// Mitsubishi GX Works2 project: UNLD LINE 4   PLC: Q06UDV

PROGRAM DATALINK
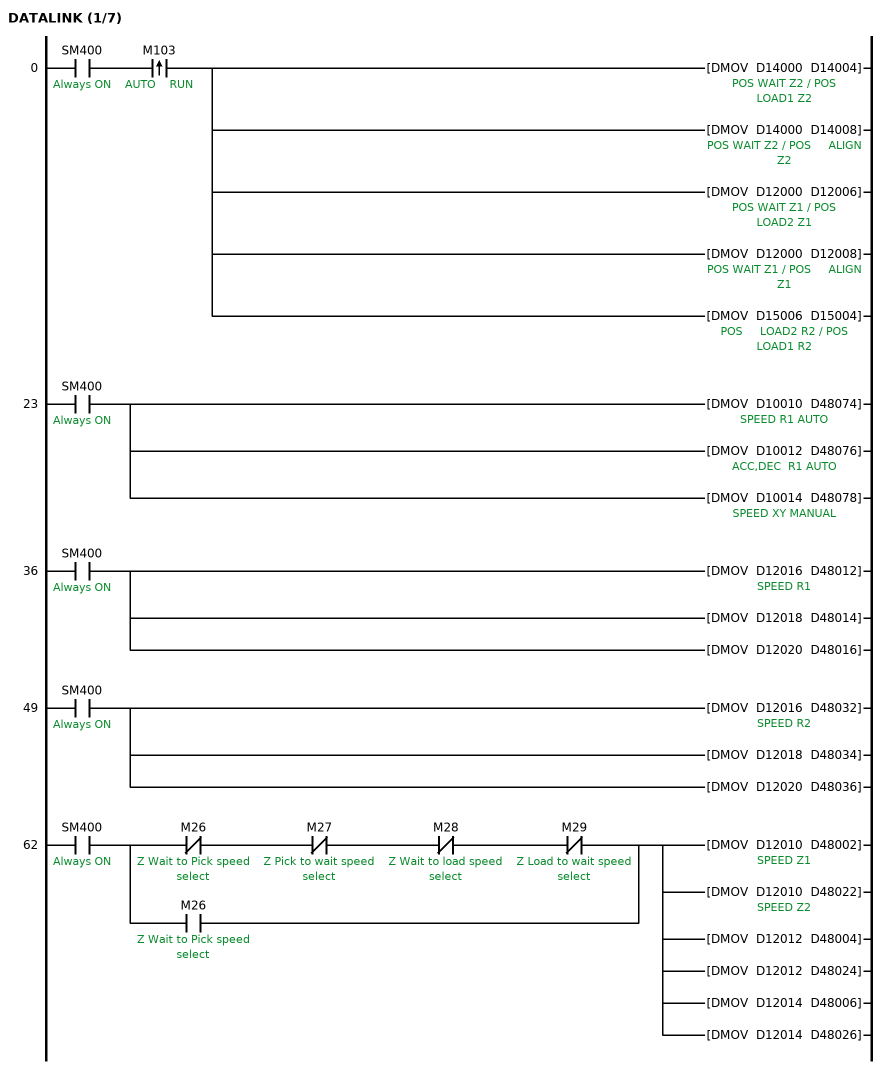
0     LD      SM400  ; Always ON
      ANDP    M103  ; AUTO    RUN
      DMOV    D14000 D14004  ; POS WAIT Z2 / POS     LOAD1 Z2
      DMOV    D14000 D14008  ; POS     ALIGN Z2
      DMOV    D12000 D12006  ; POS WAIT Z1 / POS     LOAD2 Z1
      DMOV    D12000 D12008  ; POS     ALIGN Z1
      DMOV    D15006 D15004  ; POS     LOAD2 R2 / POS     LOAD1 R2
23    LD      SM400  ; Always ON
      DMOV    D10010 D48074  ; SPEED R1 AUTO
      DMOV    D10012 D48076  ; ACC,DEC  R1 AUTO
      DMOV    D10014 D48078  ; SPEED XY MANUAL
36    LD      SM400  ; Always ON
      DMOV    D12016 D48012  ; SPEED R1
      DMOV    D12018 D48014
      DMOV    D12020 D48016
49    LD      SM400  ; Always ON
      DMOV    D12016 D48032  ; SPEED R2
      DMOV    D12018 D48034
      DMOV    D12020 D48036
62    LD      SM400  ; Always ON
      LDI     M26  ; Z Wait to Pick speed select
      ANI     M27  ; Z Pick to wait speed select
      ANI     M28  ; Z Wait to load speed select
      ANI     M29  ; Z Load to wait speed select
      OR      M26  ; Z Wait to Pick speed select
      ANB
      DMOV    D12010 D48002  ; SPEED Z1
      DMOV    D12010 D48022  ; SPEED Z2
      DMOV    D12012 D48004
      DMOV    D12012 D48024
      DMOV    D12014 D48006
      DMOV    D12014 D48026
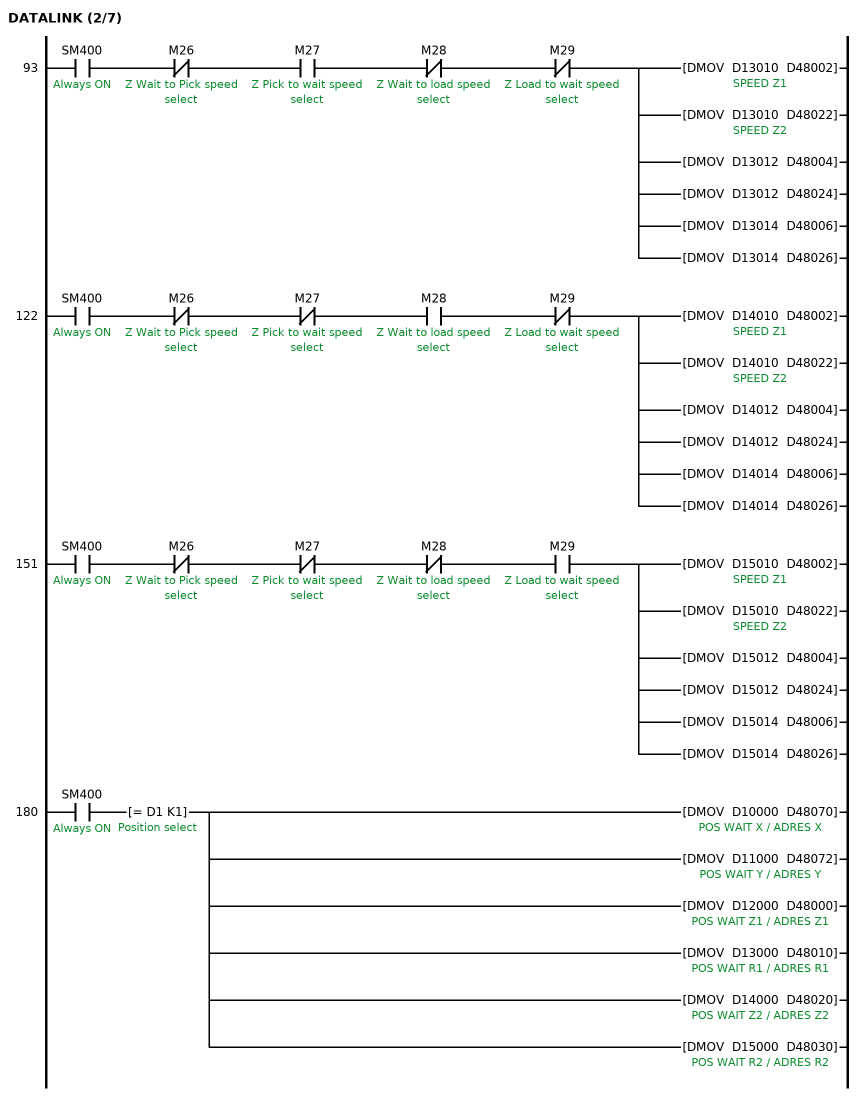
93    LD      SM400  ; Always ON
      ANI     M26  ; Z Wait to Pick speed select
      AND     M27  ; Z Pick to wait speed select
      ANI     M28  ; Z Wait to load speed select
      ANI     M29  ; Z Load to wait speed select
      DMOV    D13010 D48002
      DMOV    D13010 D48022
      DMOV    D13012 D48004
      DMOV    D13012 D48024
      DMOV    D13014 D48006
      DMOV    D13014 D48026
122   LD      SM400  ; Always ON
      ANI     M26  ; Z Wait to Pick speed select
      ANI     M27  ; Z Pick to wait speed select
      AND     M28  ; Z Wait to load speed select
      ANI     M29  ; Z Load to wait speed select
      DMOV    D14010 D48002
      DMOV    D14010 D48022
      DMOV    D14012 D48004
      DMOV    D14012 D48024
      DMOV    D14014 D48006
      DMOV    D14014 D48026
151   LD      SM400  ; Always ON
      ANI     M26  ; Z Wait to Pick speed select
      ANI     M27  ; Z Pick to wait speed select
      ANI     M28  ; Z Wait to load speed select
      AND     M29  ; Z Load to wait speed select
      DMOV    D15010 D48002
      DMOV    D15010 D48022
      DMOV    D15012 D48004
      DMOV    D15012 D48024
      DMOV    D15014 D48006
      DMOV    D15014 D48026
180   LD      SM400  ; Always ON
      AND=    D1 K1  ; Position select
      DMOV    D10000 D48070  ; POS WAIT X / ADRES X
      DMOV    D11000 D48072  ; POS WAIT Y / ADRES Y
      DMOV    D12000 D48000  ; ADRES Z1
      DMOV    D13000 D48010  ; POS WAIT R1 / ADRES R1
      DMOV    D14000 D48020  ; ADRES Z2
      DMOV    D15000 D48030  ; POS WAIT R2 / ADRES R2
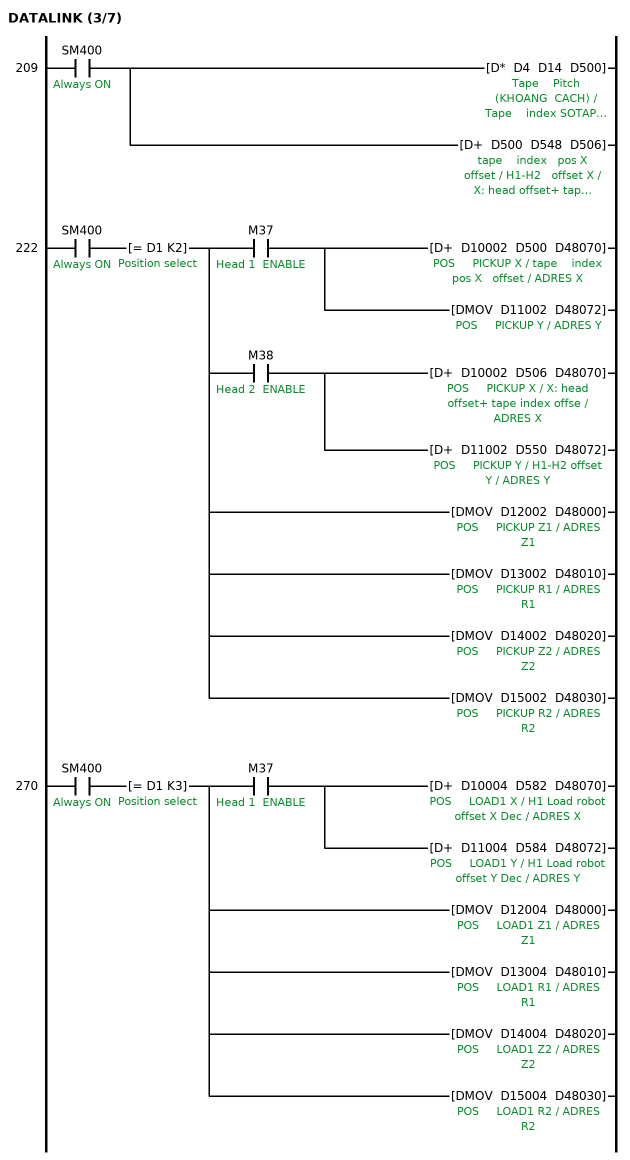
209   LD      SM400  ; Always ON
      D*      D4 D14 D500  ; Tape    Pitch   (KHOANG  CACH) / Tape    index SOTAPE HUT DUOC / tape    index   pos X   offset
      D+      D500 D548 D506  ; H1-H2   offset X / X: head offset+ tape index offse
222   LD      SM400  ; Always ON
      AND=    D1 K2  ; Position select
      MPS
      AND     M37  ; Head 1  ENABLE
      D+      D10002 D500 D48070  ; POS     PICKUP X
      DMOV    D11002 D48072  ; POS     PICKUP Y
      MRD
      AND     M38  ; Head 2  ENABLE
      D+      D10002 D506 D48070
      D+      D11002 D550 D48072  ; H1-H2 offset Y
      MPP
      DMOV    D12002 D48000  ; POS     PICKUP Z1
      DMOV    D13002 D48010  ; POS     PICKUP R1
      DMOV    D14002 D48020  ; POS     PICKUP Z2
      DMOV    D15002 D48030  ; POS     PICKUP R2
270   LD      SM400  ; Always ON
      AND=    D1 K3  ; Position select
      MPS
      AND     M37  ; Head 1  ENABLE
      D+      D10004 D582 D48070  ; POS     LOAD1 X / H1 Load robot offset X Dec
      D+      D11004 D584 D48072  ; POS     LOAD1 Y / H1 Load robot offset Y Dec
      MPP
      DMOV    D12004 D48000  ; POS     LOAD1 Z1
      DMOV    D13004 D48010  ; POS     LOAD1 R1
      DMOV    D14004 D48020
      DMOV    D15004 D48030
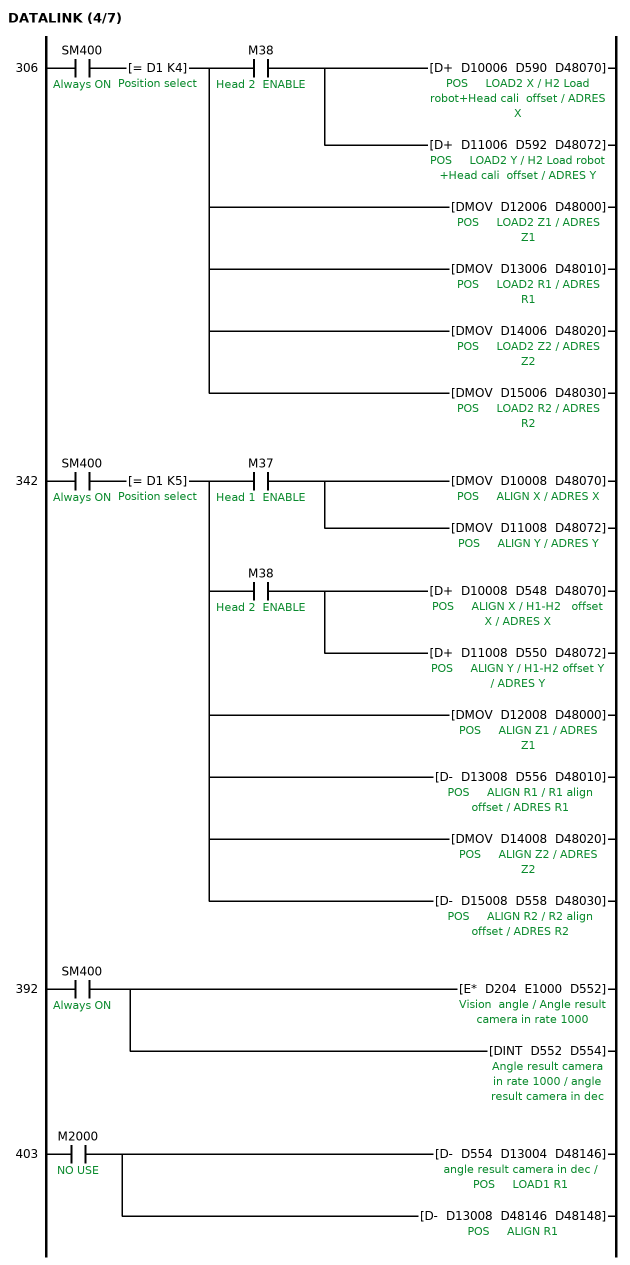
306   LD      SM400  ; Always ON
      AND=    D1 K4  ; Position select
      MPS
      AND     M38  ; Head 2  ENABLE
      D+      D10006 D590 D48070  ; POS     LOAD2 X / H2 Load robot+Head cali  offset
      D+      D11006 D592 D48072  ; POS     LOAD2 Y / H2 Load robot +Head cali  offset
      MPP
      DMOV    D12006 D48000
      DMOV    D13006 D48010  ; POS     LOAD2 R1
      DMOV    D14006 D48020  ; POS     LOAD2 Z2
      DMOV    D15006 D48030
342   LD      SM400  ; Always ON
      AND=    D1 K5  ; Position select
      MPS
      AND     M37  ; Head 1  ENABLE
      DMOV    D10008 D48070  ; POS     ALIGN X
      DMOV    D11008 D48072  ; POS     ALIGN Y
      MRD
      AND     M38  ; Head 2  ENABLE
      D+      D10008 D548 D48070
      D+      D11008 D550 D48072
      MPP
      DMOV    D12008 D48000
      D-      D13008 D556 D48010  ; POS     ALIGN R1 / R1 align offset
      DMOV    D14008 D48020
      D-      D15008 D558 D48030  ; POS     ALIGN R2 / R2 align offset
392   LD      SM400  ; Always ON
      E*      D204 E1000 D552  ; Vision  angle / Angle result camera in rate 1000
      DINT    D552 D554  ; angle result camera in dec
403   LD      M2000  ; NO USE
      D-      D554 D13004 D48146
      D-      D13008 D48146 D48148
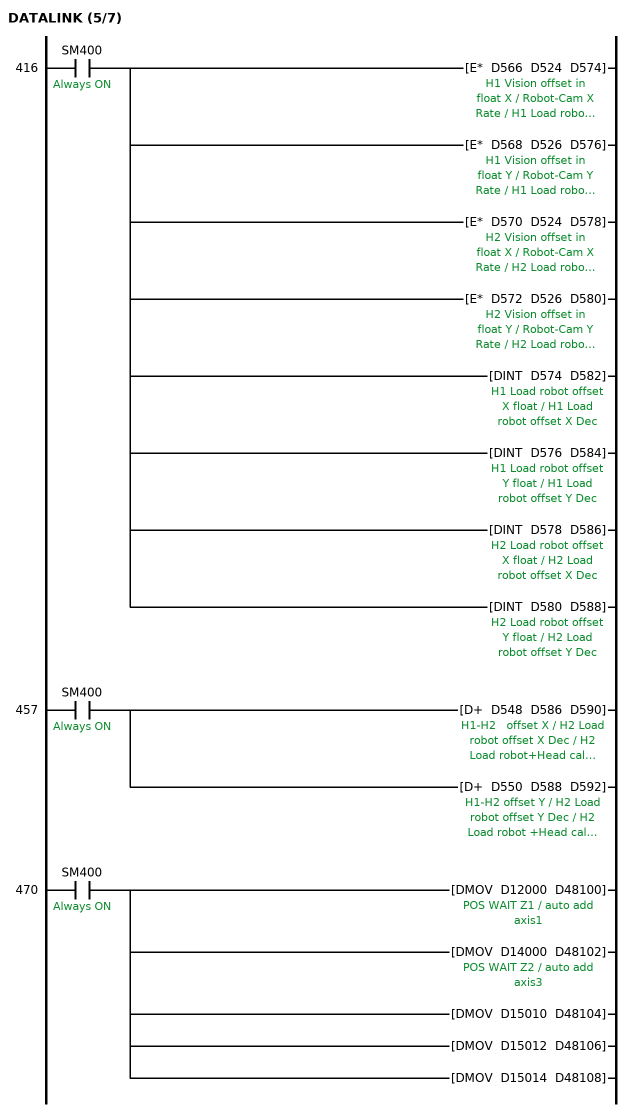
416   LD      SM400  ; Always ON
      E*      D566 D524 D574  ; H1 Vision offset in     float X / Robot-Cam X Rate / H1 Load robot offset X float
      E*      D568 D526 D576  ; H1 Vision offset in     float Y / Robot-Cam Y Rate / H1 Load robot offset Y float
      E*      D570 D524 D578  ; H2 Vision offset in     float X / H2 Load robot offset X float
      E*      D572 D526 D580  ; H2 Vision offset in     float Y / H2 Load robot offset Y float
      DINT    D574 D582
      DINT    D576 D584
      DINT    D578 D586  ; H2 Load robot offset X Dec
      DINT    D580 D588  ; H2 Load robot offset Y Dec
457   LD      SM400  ; Always ON
      D+      D548 D586 D590
      D+      D550 D588 D592
470   LD      SM400  ; Always ON
      DMOV    D12000 D48100  ; auto add axis1
      DMOV    D14000 D48102  ; auto add axis3
      DMOV    D15010 D48104
      DMOV    D15012 D48106
      DMOV    D15014 D48108
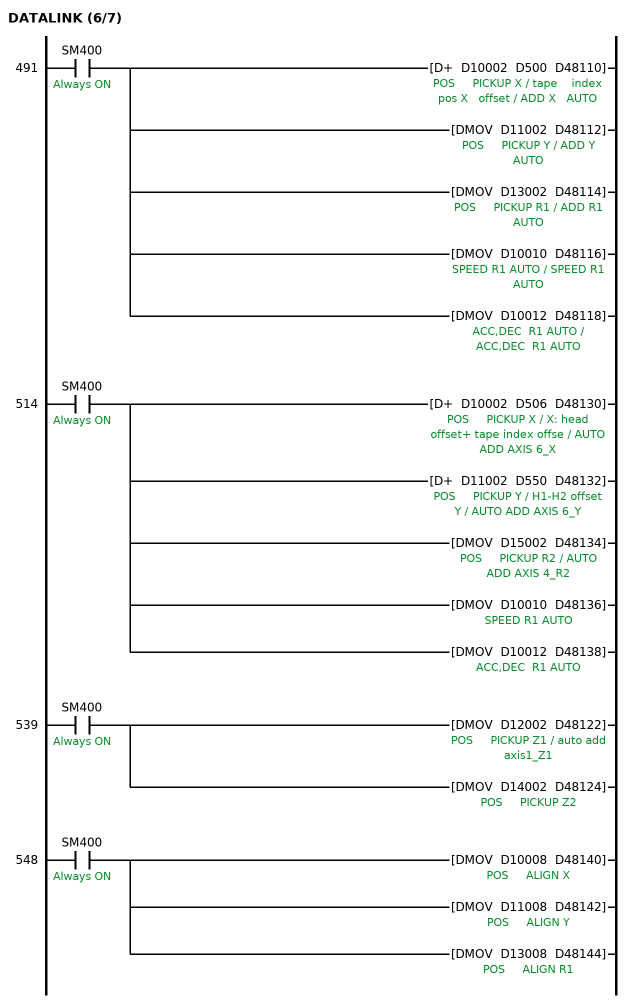
491   LD      SM400  ; Always ON
      D+      D10002 D500 D48110  ; ADD X   AUTO
      DMOV    D11002 D48112  ; ADD Y   AUTO
      DMOV    D13002 D48114  ; ADD R1  AUTO
      DMOV    D10010 D48116  ; SPEED R1 AUTO
      DMOV    D10012 D48118  ; ACC,DEC  R1 AUTO
514   LD      SM400  ; Always ON
      D+      D10002 D506 D48130  ; AUTO ADD AXIS 6_X
      D+      D11002 D550 D48132  ; AUTO ADD AXIS 6_Y
      DMOV    D15002 D48134  ; AUTO ADD AXIS 4_R2
      DMOV    D10010 D48136
      DMOV    D10012 D48138
539   LD      SM400  ; Always ON
      DMOV    D12002 D48122  ; auto add axis1_Z1
      DMOV    D14002 D48124
548   LD      SM400  ; Always ON
      DMOV    D10008 D48140
      DMOV    D11008 D48142
      DMOV    D13008 D48144
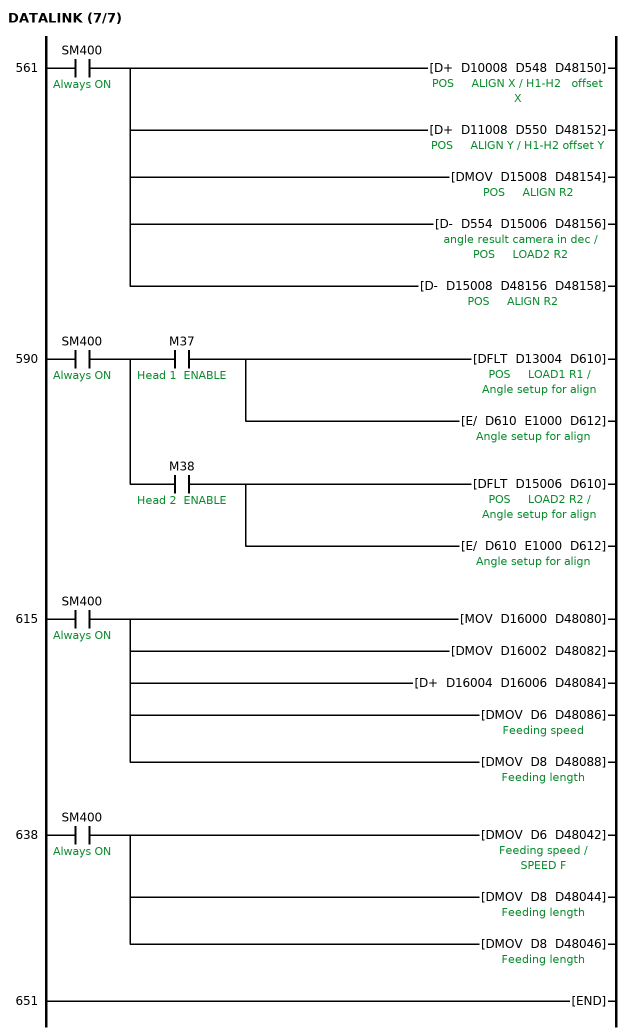
561   LD      SM400  ; Always ON
      D+      D10008 D548 D48150
      D+      D11008 D550 D48152
      DMOV    D15008 D48154
      D-      D554 D15006 D48156
      D-      D15008 D48156 D48158
590   LD      SM400  ; Always ON
      MPS
      AND     M37  ; Head 1  ENABLE
      DFLT    D13004 D610  ; Angle setup for align
      E/      D610 E1000 D612
      MPP
      AND     M38  ; Head 2  ENABLE
      DFLT    D15006 D610
      E/      D610 E1000 D612
615   LD      SM400  ; Always ON
      MOV     D16000 D48080
      DMOV    D16002 D48082
      D+      D16004 D16006 D48084
      DMOV    D6 D48086  ; Feeding speed
      DMOV    D8 D48088  ; Feeding length
638   LD      SM400  ; Always ON
      DMOV    D6 D48042  ; SPEED F
      DMOV    D8 D48044
      DMOV    D8 D48046
651   END
END_PROGRAM

PROGRAM MAIN
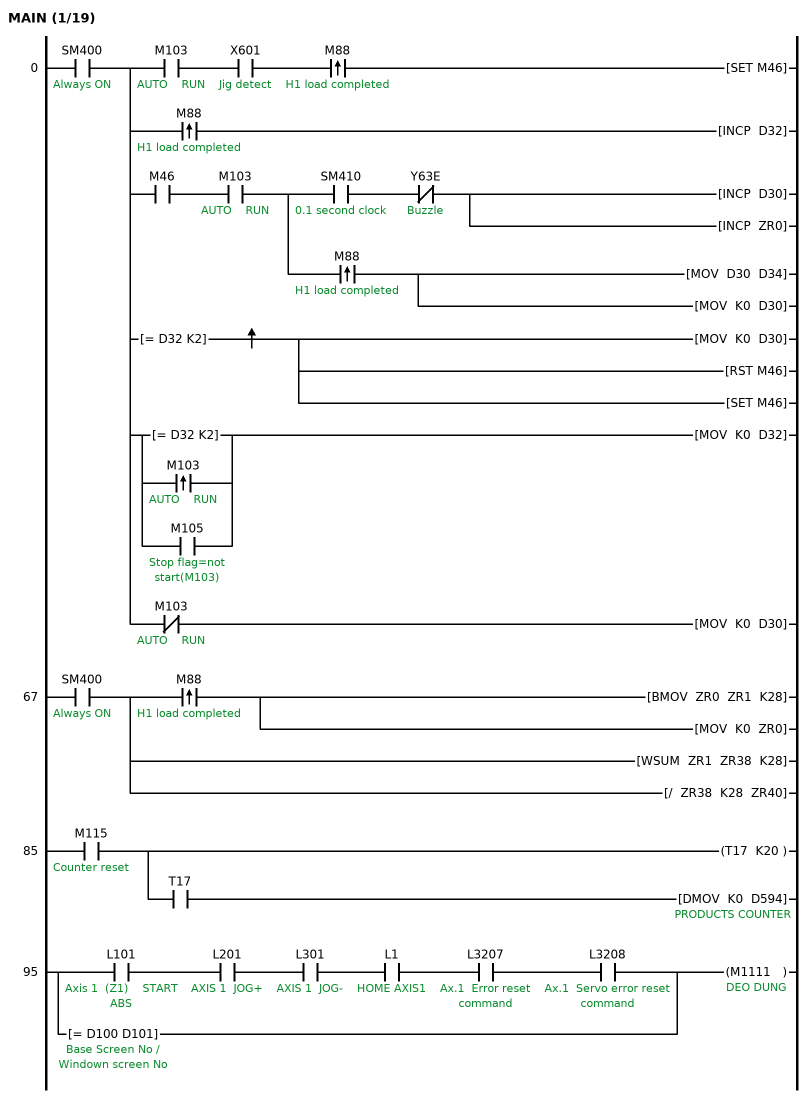
0     LD      SM400  ; Always ON
      MPS
      AND     M103  ; AUTO    RUN
      AND     X601  ; Jig detect
      ANDP    M88  ; H1 load completed
      SET     M46
      MRD
      ANDP    M88  ; H1 load completed
      INCP    D32
      MRD
      AND     M46
      AND     M103  ; AUTO    RUN
      MPS
      AND     SM410  ; 0.1 second clock
      ANI     Y63E  ; Buzzle
      INCP    D30
      INCP    ZR0
      MPP
      ANDP    M88  ; H1 load completed
      MOV     D30 D34
      MOV     K0 D30
      MRD
      AND=    D32 K2
      MEP
      MOV     K0 D30
      RST     M46
      SET     M46
      MRD
      LD=     D32 K2
      ORP     M103  ; AUTO    RUN
      OR      M105  ; Stop flag=not start(M103)
      ANB
      MOV     K0 D32
      MPP
      ANI     M103  ; AUTO    RUN
      MOV     K0 D30
67    LD      SM400  ; Always ON
      MPS
      ANDP    M88  ; H1 load completed
      BMOV    ZR0 ZR1 K28
      MOV     K0 ZR0
      MPP
      WSUM    ZR1 ZR38 K28
      /       ZR38 K28 ZR40
85    LD      M115  ; Counter reset
      OUT     T17 K20
      AND     T17
      DMOV    K0 D594  ; PRODUCTS COUNTER
95    LD      L101  ; Axis 1  (Z1)    START   ABS
      AND     L201  ; AXIS 1  JOG+
      AND     L301  ; AXIS 1  JOG-
      AND     L1  ; HOME AXIS1
      AND     L3207  ; Ax.1  Error reset command
      AND     L3208  ; Ax.1  Servo error reset command
      OR=     D100 D101  ; Base Screen No / Windown screen No
      OUT     M1111  ; DEO DUNG
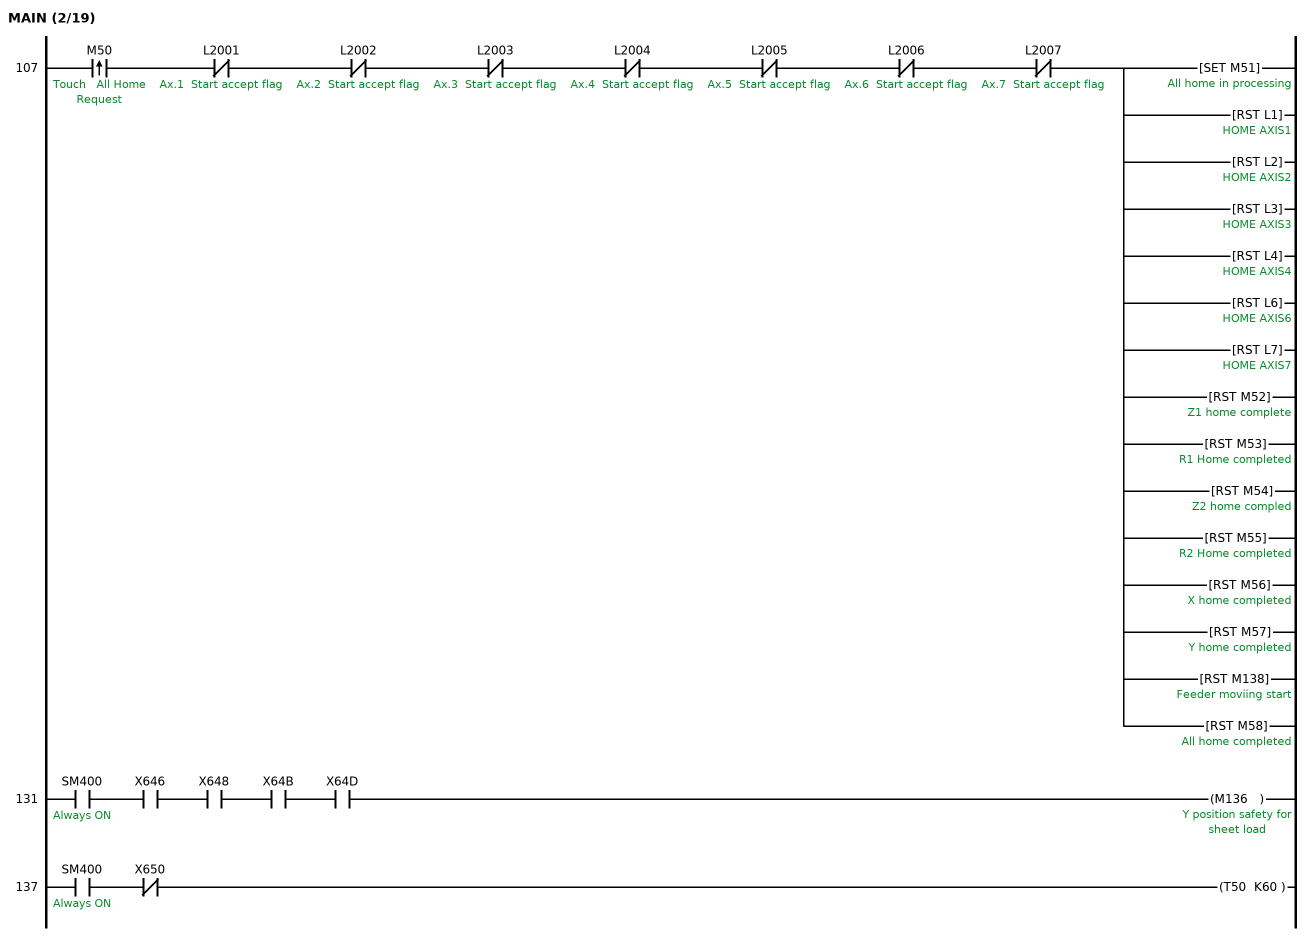
107   LDP     M50  ; Touch   All Home Request
      ANI     L2001  ; Ax.1  Start accept flag
      ANI     L2002  ; Ax.2  Start accept flag
      ANI     L2003  ; Ax.3  Start accept flag
      ANI     L2004  ; Ax.4  Start accept flag
      ANI     L2005  ; Ax.5  Start accept flag
      ANI     L2006  ; Ax.6  Start accept flag
      ANI     L2007  ; Ax.7  Start accept flag
      SET     M51  ; All home in processing
      RST     L1  ; HOME AXIS1
      RST     L2  ; HOME AXIS2
      RST     L3  ; HOME AXIS3
      RST     L4  ; HOME AXIS4
      RST     L6  ; HOME AXIS6
      RST     L7  ; HOME AXIS7
      RST     M52  ; Z1 home complete
      RST     M53  ; R1 Home completed
      RST     M54  ; Z2 home compled
      RST     M55  ; R2 Home completed
      RST     M56  ; X home completed
      RST     M57  ; Y home completed
      RST     M138  ; Feeder moviing start
      RST     M58  ; All home completed
131   LD      SM400  ; Always ON
      AND     X646
      AND     X648
      AND     X64B
      AND     X64D
      OUT     M136  ; Y position safety for sheet load
137   LD      SM400  ; Always ON
      ANI     X650
      OUT     T50 K60
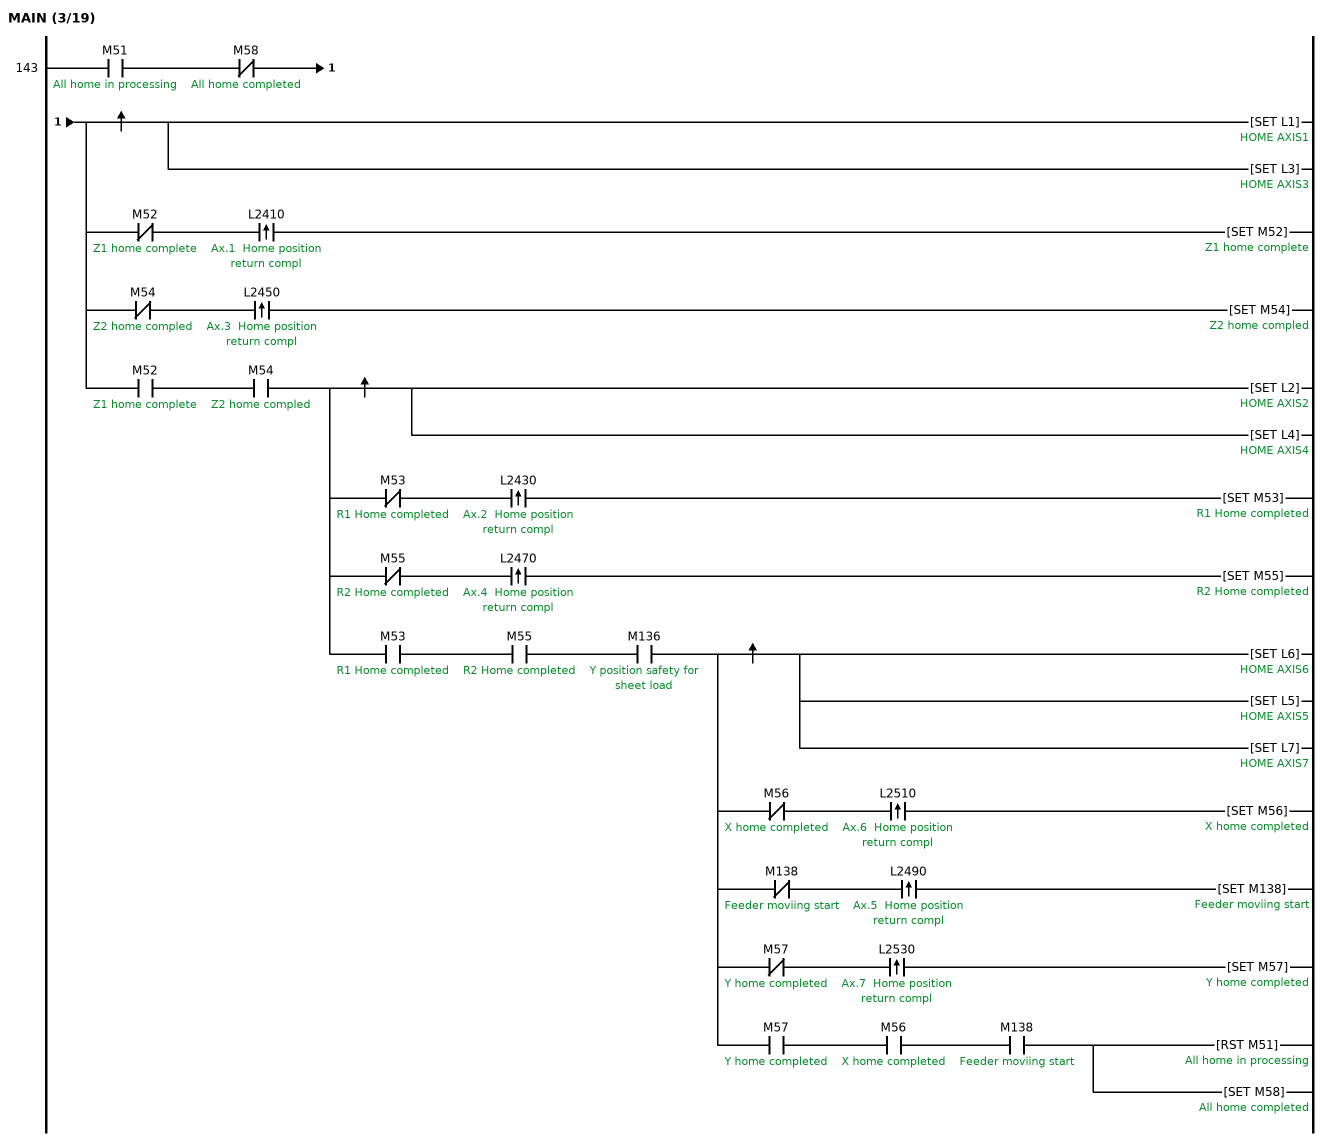
143   LD      M51  ; All home in processing
      ANI     M58  ; All home completed
      MPS
      MEP
      SET     L1  ; HOME AXIS1
      SET     L3  ; HOME AXIS3
      MRD
      ANI     M52  ; Z1 home complete
      ANDP    L2410  ; Ax.1  Home position return compl
      SET     M52  ; Z1 home complete
      MRD
      ANI     M54  ; Z2 home compled
      ANDP    L2450  ; Ax.3  Home position return compl
      SET     M54  ; Z2 home compled
      MPP
      AND     M52  ; Z1 home complete
      AND     M54  ; Z2 home compled
      MPS
      MEP
      SET     L2  ; HOME AXIS2
      SET     L4  ; HOME AXIS4
      MRD
      ANI     M53  ; R1 Home completed
      ANDP    L2430  ; Ax.2  Home position return compl
      SET     M53  ; R1 Home completed
      MRD
      ANI     M55  ; R2 Home completed
      ANDP    L2470  ; Ax.4  Home position return compl
      SET     M55  ; R2 Home completed
      MPP
      AND     M53  ; R1 Home completed
      AND     M55  ; R2 Home completed
      AND     M136  ; Y position safety for sheet load
      MPS
      MEP
      SET     L6  ; HOME AXIS6
      SET     L5  ; HOME AXIS5
      SET     L7  ; HOME AXIS7
      MRD
      ANI     M56  ; X home completed
      ANDP    L2510  ; Ax.6  Home position return compl
      SET     M56  ; X home completed
      MRD
      ANI     M138  ; Feeder moviing start
      ANDP    L2490  ; Ax.5  Home position return compl
      SET     M138  ; Feeder moviing start
      MRD
      ANI     M57  ; Y home completed
      ANDP    L2530  ; Ax.7  Home position return compl
      SET     M57  ; Y home completed
      MPP
      AND     M57  ; Y home completed
      AND     M56  ; X home completed
      AND     M138  ; Feeder moviing start
      RST     M51  ; All home in processing
      SET     M58  ; All home completed
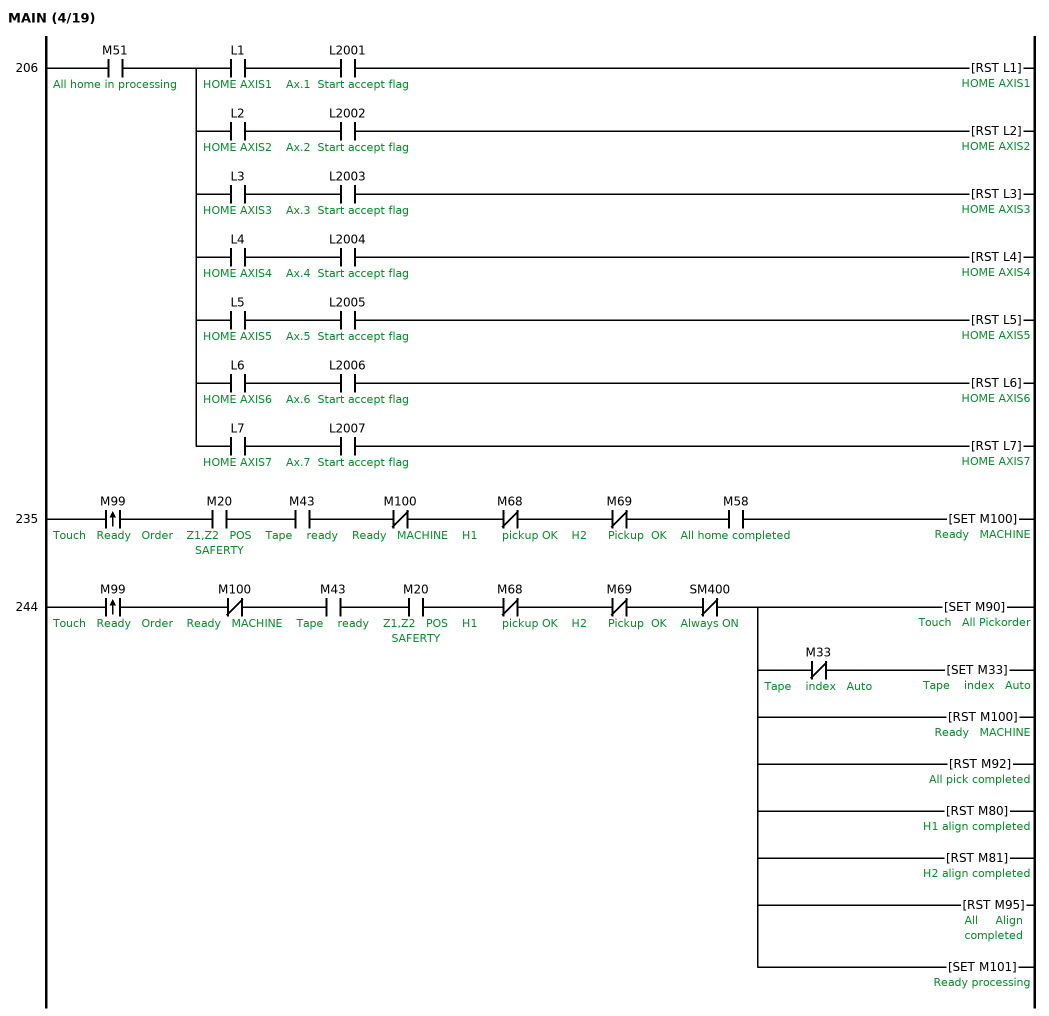
206   LD      M51  ; All home in processing
      MPS
      AND     L1  ; HOME AXIS1
      AND     L2001  ; Ax.1  Start accept flag
      RST     L1  ; HOME AXIS1
      MRD
      AND     L2  ; HOME AXIS2
      AND     L2002  ; Ax.2  Start accept flag
      RST     L2  ; HOME AXIS2
      MRD
      AND     L3  ; HOME AXIS3
      AND     L2003  ; Ax.3  Start accept flag
      RST     L3  ; HOME AXIS3
      MRD
      AND     L4  ; HOME AXIS4
      AND     L2004  ; Ax.4  Start accept flag
      RST     L4  ; HOME AXIS4
      MRD
      AND     L5  ; HOME AXIS5
      AND     L2005  ; Ax.5  Start accept flag
      RST     L5  ; HOME AXIS5
      MRD
      AND     L6  ; HOME AXIS6
      AND     L2006  ; Ax.6  Start accept flag
      RST     L6  ; HOME AXIS6
      MPP
      AND     L7  ; HOME AXIS7
      AND     L2007  ; Ax.7  Start accept flag
      RST     L7  ; HOME AXIS7
235   LDP     M99  ; Touch   Ready   Order
      AND     M20  ; Z1,Z2   POS     SAFERTY
      AND     M43  ; Tape    ready
      ANI     M100  ; Ready   MACHINE
      ANI     M68  ; H1       pickup OK
      ANI     M69  ; H2      Pickup  OK
      AND     M58  ; All home completed
      SET     M100  ; Ready   MACHINE
244   LDP     M99  ; Touch   Ready   Order
      ANI     M100  ; Ready   MACHINE
      AND     M43  ; Tape    ready
      AND     M20  ; Z1,Z2   POS     SAFERTY
      ANI     M68  ; H1       pickup OK
      ANI     M69  ; H2      Pickup  OK
      ANI     SM400  ; Always ON
      SET     M90  ; Touch   All Pickorder
      MPS
      ANI     M33  ; Tape    index   Auto
      SET     M33  ; Tape    index   Auto
      MPP
      RST     M100  ; Ready   MACHINE
      RST     M92  ; All pick completed
      RST     M80  ; H1 align completed
      RST     M81  ; H2 align completed
      RST     M95  ; All     Align   completed
      SET     M101  ; Ready processing
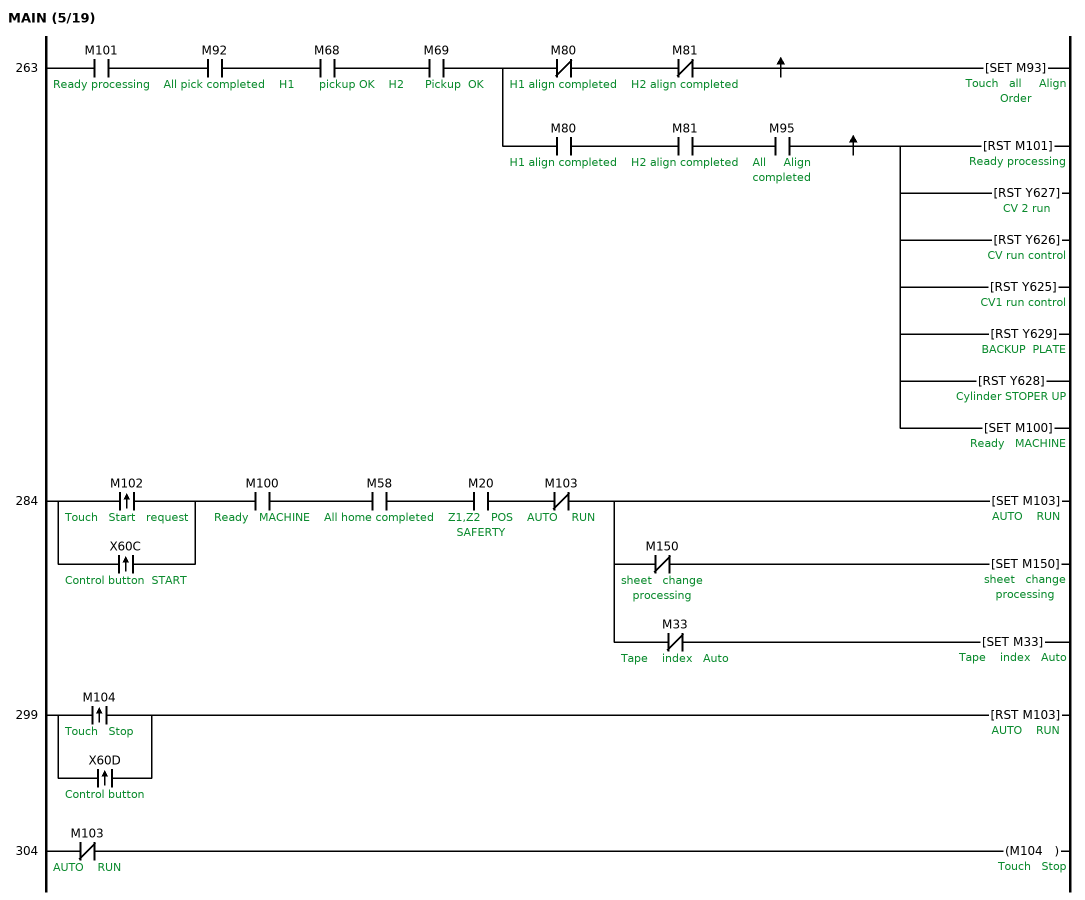
263   LD      M101  ; Ready processing
      AND     M92  ; All pick completed
      AND     M68  ; H1       pickup OK
      AND     M69  ; H2      Pickup  OK
      MPS
      ANI     M80  ; H1 align completed
      ANI     M81  ; H2 align completed
      MEP
      SET     M93  ; Touch   all     Align   Order
      MPP
      AND     M80  ; H1 align completed
      AND     M81  ; H2 align completed
      AND     M95  ; All     Align   completed
      MEP
      RST     M101  ; Ready processing
      RST     Y627  ; CV 2 run
      RST     Y626  ; CV run control
      RST     Y625  ; CV1 run control
      RST     Y629  ; BACKUP  PLATE
      RST     Y628  ; Cylinder STOPER UP
      SET     M100  ; Ready   MACHINE
284   LDP     M102  ; Touch   Start   request
      ORP     X60C  ; Control button  START
      AND     M100  ; Ready   MACHINE
      AND     M58  ; All home completed
      AND     M20  ; Z1,Z2   POS     SAFERTY
      ANI     M103  ; AUTO    RUN
      SET     M103  ; AUTO    RUN
      MPS
      ANI     M150  ; sheet   change  processing
      SET     M150  ; sheet   change  processing
      MPP
      ANI     M33  ; Tape    index   Auto
      SET     M33  ; Tape    index   Auto
299   LDP     M104  ; Touch   Stop
      ORP     X60D  ; Control button
      RST     M103  ; AUTO    RUN
304   LDI     M103  ; AUTO    RUN
      OUT     M104  ; Touch   Stop
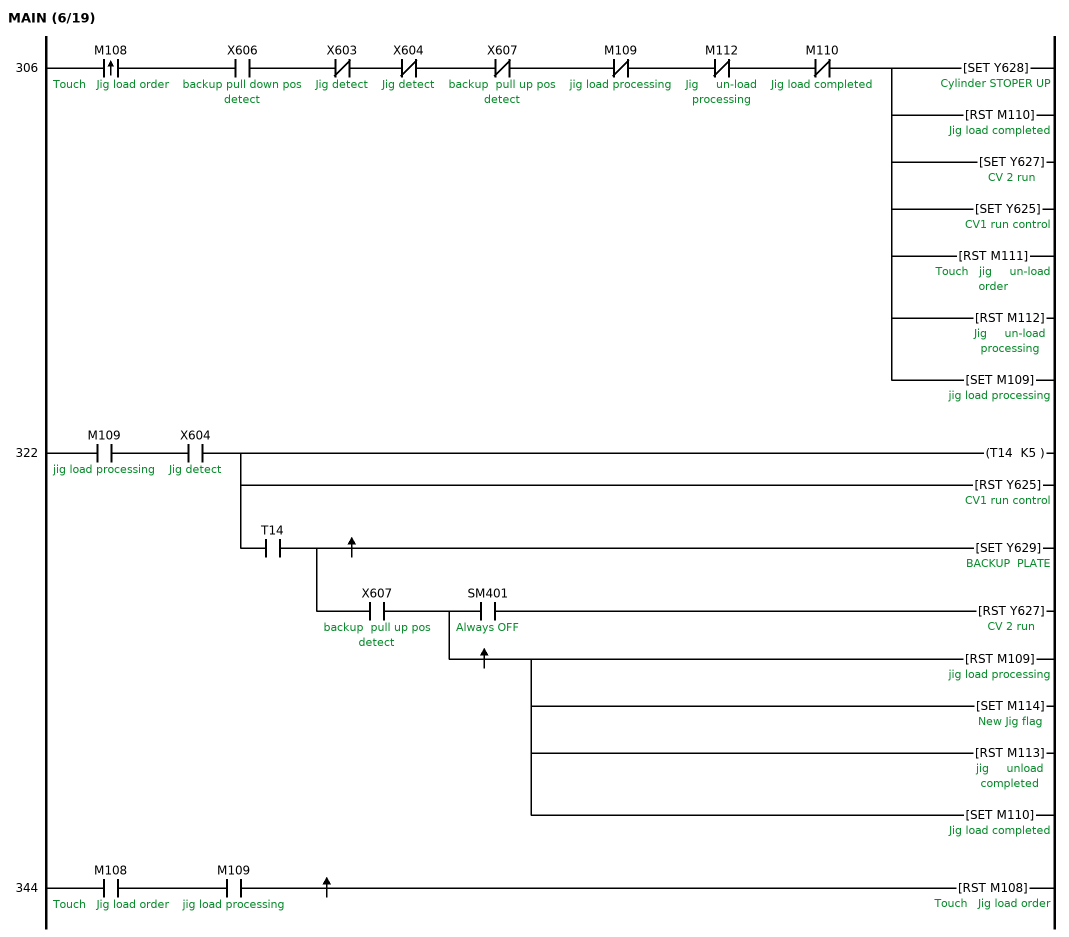
306   LDP     M108  ; Touch   Jig load order
      AND     X606  ; backup pull down pos detect
      ANI     X603  ; Jig detect
      ANI     X604  ; Jig detect
      ANI     X607  ; backup  pull up pos     detect
      ANI     M109  ; jig load processing
      ANI     M112  ; Jig     un-load processing
      ANI     M110  ; Jig load completed
      SET     Y628  ; Cylinder STOPER UP
      RST     M110  ; Jig load completed
      SET     Y627  ; CV 2 run
      SET     Y625  ; CV1 run control
      RST     M111  ; Touch   jig     un-load order
      RST     M112  ; Jig     un-load processing
      SET     M109  ; jig load processing
322   LD      M109  ; jig load processing
      AND     X604  ; Jig detect
      OUT     T14 K5
      RST     Y625  ; CV1 run control
      AND     T14
      MPS
      MEP
      SET     Y629  ; BACKUP  PLATE
      MPP
      AND     X607  ; backup  pull up pos     detect
      MPS
      AND     SM401  ; Always OFF
      RST     Y627  ; CV 2 run
      MPP
      MEP
      RST     M109  ; jig load processing
      SET     M114  ; New Jig flag
      RST     M113  ; jig     unload  completed
      SET     M110  ; Jig load completed
344   LD      M108  ; Touch   Jig load order
      AND     M109  ; jig load processing
      MEP
      RST     M108  ; Touch   Jig load order
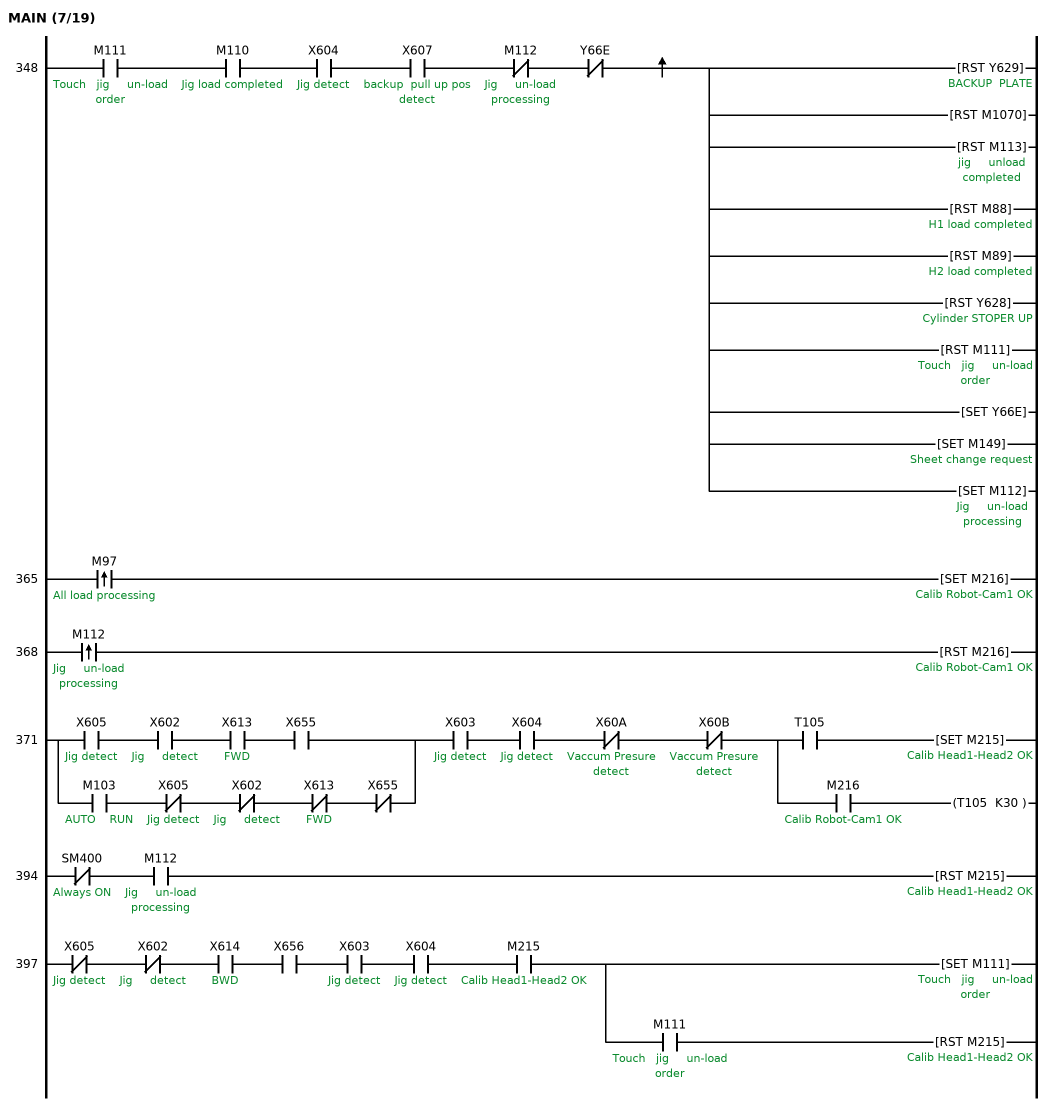
348   LD      M111  ; Touch   jig     un-load order
      AND     M110  ; Jig load completed
      AND     X604  ; Jig detect
      AND     X607  ; backup  pull up pos     detect
      ANI     M112  ; Jig     un-load processing
      ANI     Y66E
      MEP
      RST     Y629  ; BACKUP  PLATE
      RST     M1070
      RST     M113  ; jig     unload  completed
      RST     M88  ; H1 load completed
      RST     M89  ; H2 load completed
      RST     Y628  ; Cylinder STOPER UP
      RST     M111  ; Touch   jig     un-load order
      SET     Y66E
      SET     M149  ; Sheet change request
      SET     M112  ; Jig     un-load processing
365   LDP     M97  ; All load processing
      SET     M216  ; Calib Robot-Cam1 OK
368   LDP     M112  ; Jig     un-load processing
      RST     M216  ; Calib Robot-Cam1 OK
371   LD      X605  ; Jig detect
      AND     X602  ; Jig     detect
      AND     X613  ; FWD
      AND     X655
      LD      M103  ; AUTO    RUN
      ANI     X605  ; Jig detect
      ANI     X602  ; Jig     detect
      ANI     X613  ; FWD
      ANI     X655
      ORB
      AND     X603  ; Jig detect
      AND     X604  ; Jig detect
      ANI     X60A  ; Vaccum Presure detect
      ANI     X60B  ; Vaccum Presure detect
      MPS
      AND     T105
      SET     M215  ; Calib Head1-Head2 OK
      MPP
      AND     M216  ; Calib Robot-Cam1 OK
      OUT     T105 K30
394   LDI     SM400  ; Always ON
      AND     M112  ; Jig     un-load processing
      RST     M215  ; Calib Head1-Head2 OK
397   LDI     X605  ; Jig detect
      ANI     X602  ; Jig     detect
      AND     X614  ; BWD
      AND     X656
      AND     X603  ; Jig detect
      AND     X604  ; Jig detect
      AND     M215  ; Calib Head1-Head2 OK
      SET     M111  ; Touch   jig     un-load order
      AND     M111  ; Touch   jig     un-load order
      RST     M215  ; Calib Head1-Head2 OK
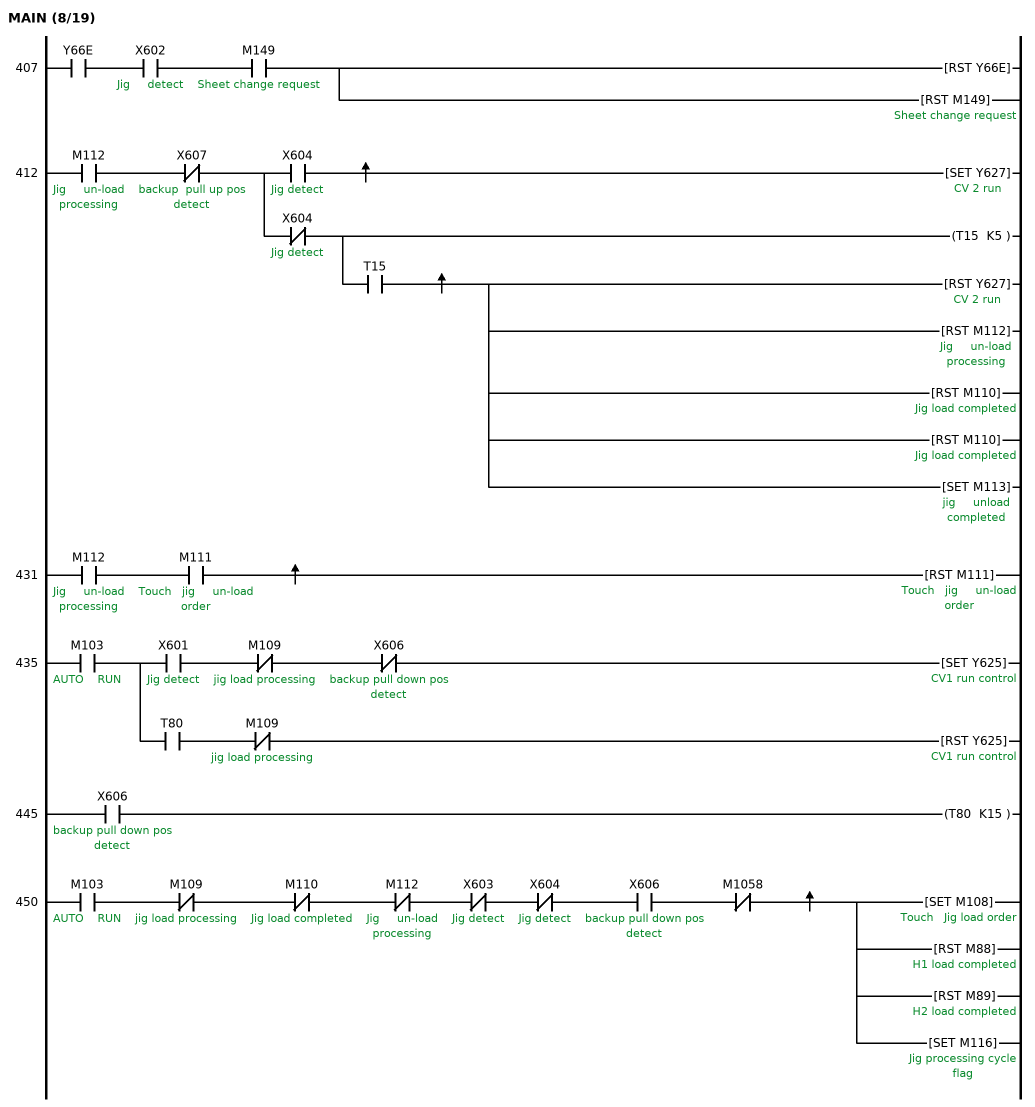
407   LD      Y66E
      AND     X602  ; Jig     detect
      AND     M149  ; Sheet change request
      RST     Y66E
      RST     M149  ; Sheet change request
412   LD      M112  ; Jig     un-load processing
      ANI     X607  ; backup  pull up pos     detect
      MPS
      AND     X604  ; Jig detect
      MEP
      SET     Y627  ; CV 2 run
      MPP
      ANI     X604  ; Jig detect
      OUT     T15 K5
      AND     T15
      MEP
      RST     Y627  ; CV 2 run
      RST     M112  ; Jig     un-load processing
      RST     M110  ; Jig load completed
      RST     M110  ; Jig load completed
      SET     M113  ; jig     unload  completed
431   LD      M112  ; Jig     un-load processing
      AND     M111  ; Touch   jig     un-load order
      MEP
      RST     M111  ; Touch   jig     un-load order
435   LD      M103  ; AUTO    RUN
      MPS
      AND     X601  ; Jig detect
      ANI     M109  ; jig load processing
      ANI     X606  ; backup pull down pos detect
      SET     Y625  ; CV1 run control
      MPP
      AND     T80
      ANI     M109  ; jig load processing
      RST     Y625  ; CV1 run control
445   LD      X606  ; backup pull down pos detect
      OUT     T80 K15
450   LD      M103  ; AUTO    RUN
      ANI     M109  ; jig load processing
      ANI     M110  ; Jig load completed
      ANI     M112  ; Jig     un-load processing
      ANI     X603  ; Jig detect
      ANI     X604  ; Jig detect
      AND     X606  ; backup pull down pos detect
      ANI     M1058
      MEP
      SET     M108  ; Touch   Jig load order
      RST     M88  ; H1 load completed
      RST     M89  ; H2 load completed
      SET     M116  ; Jig processing cycle flag
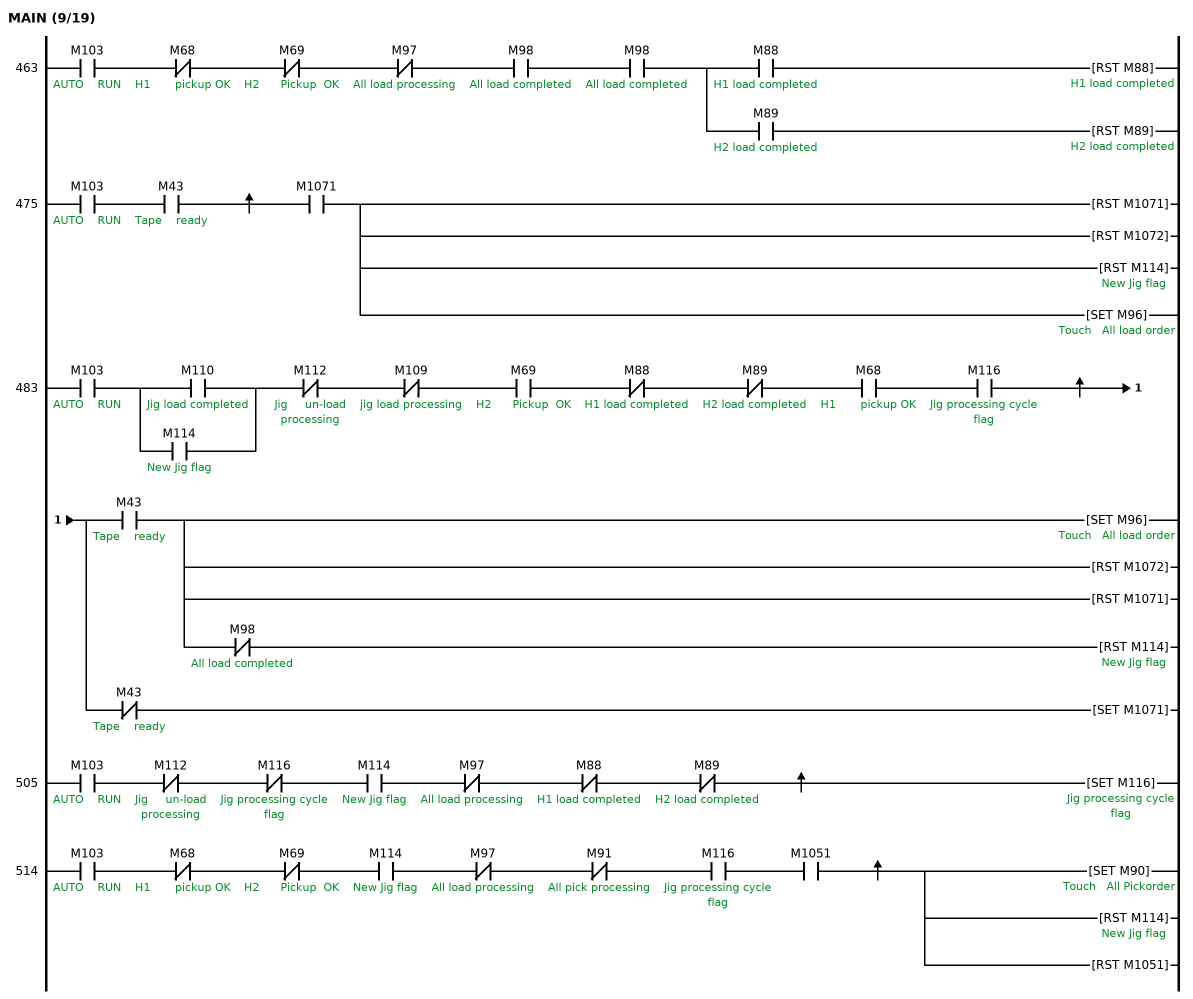
463   LD      M103  ; AUTO    RUN
      ANI     M68  ; H1       pickup OK
      ANI     M69  ; H2      Pickup  OK
      ANI     M97  ; All load processing
      AND     M98  ; All load completed
      AND     M98  ; All load completed
      MPS
      AND     M88  ; H1 load completed
      RST     M88  ; H1 load completed
      MPP
      AND     M89  ; H2 load completed
      RST     M89  ; H2 load completed
475   LD      M103  ; AUTO    RUN
      AND     M43  ; Tape    ready
      MEP
      AND     M1071
      RST     M1071
      RST     M1072
      RST     M114  ; New Jig flag
      SET     M96  ; Touch   All load order
483   LD      M103  ; AUTO    RUN
      LD      M110  ; Jig load completed
      OR      M114  ; New Jig flag
      ANB
      ANI     M112  ; Jig     un-load processing
      ANI     M109  ; jig load processing
      AND     M69  ; H2      Pickup  OK
      ANI     M88  ; H1 load completed
      ANI     M89  ; H2 load completed
      AND     M68  ; H1       pickup OK
      AND     M116  ; Jig processing cycle flag
      MEP
      MPS
      AND     M43  ; Tape    ready
      SET     M96  ; Touch   All load order
      RST     M1072
      RST     M1071
      ANI     M98  ; All load completed
      RST     M114  ; New Jig flag
      MPP
      ANI     M43  ; Tape    ready
      SET     M1071
505   LD      M103  ; AUTO    RUN
      ANI     M112  ; Jig     un-load processing
      ANI     M116  ; Jig processing cycle flag
      AND     M114  ; New Jig flag
      ANI     M97  ; All load processing
      ANI     M88  ; H1 load completed
      ANI     M89  ; H2 load completed
      MEP
      SET     M116  ; Jig processing cycle flag
514   LD      M103  ; AUTO    RUN
      ANI     M68  ; H1       pickup OK
      ANI     M69  ; H2      Pickup  OK
      AND     M114  ; New Jig flag
      ANI     M97  ; All load processing
      ANI     M91  ; All pick processing
      AND     M116  ; Jig processing cycle flag
      AND     M1051
      MEP
      SET     M90  ; Touch   All Pickorder
      RST     M114  ; New Jig flag
      RST     M1051
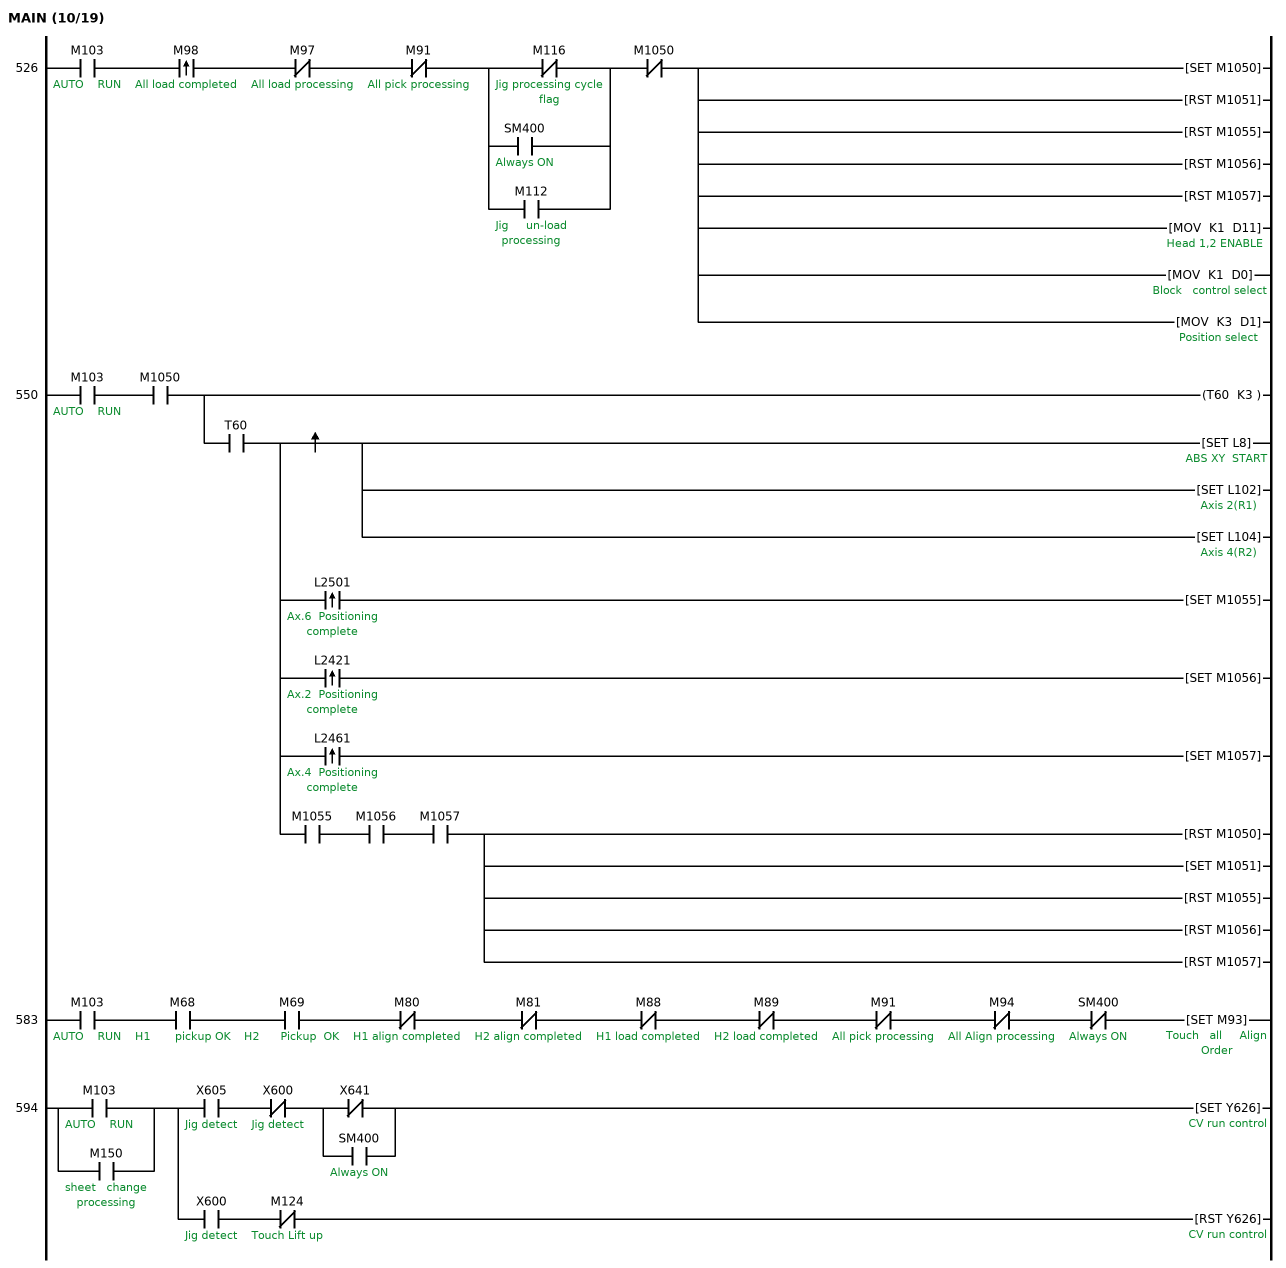
526   LD      M103  ; AUTO    RUN
      ANDP    M98  ; All load completed
      ANI     M97  ; All load processing
      ANI     M91  ; All pick processing
      LDI     M116  ; Jig processing cycle flag
      OR      SM400  ; Always ON
      OR      M112  ; Jig     un-load processing
      ANB
      ANI     M1050
      SET     M1050
      RST     M1051
      RST     M1055
      RST     M1056
      RST     M1057
      MOV     K1 D11  ; Head 1,2 ENABLE
      MOV     K1 D0  ; Block   control select
      MOV     K3 D1  ; Position select
550   LD      M103  ; AUTO    RUN
      AND     M1050
      OUT     T60 K3
      AND     T60
      MPS
      MEP
      SET     L8  ; ABS XY  START
      SET     L102  ; Axis 2(R1)
      SET     L104  ; Axis 4(R2)
      MRD
      ANDP    L2501  ; Ax.6  Positioning complete
      SET     M1055
      MRD
      ANDP    L2421  ; Ax.2  Positioning complete
      SET     M1056
      MRD
      ANDP    L2461  ; Ax.4  Positioning complete
      SET     M1057
      MPP
      AND     M1055
      AND     M1056
      AND     M1057
      RST     M1050
      SET     M1051
      RST     M1055
      RST     M1056
      RST     M1057
583   LD      M103  ; AUTO    RUN
      AND     M68  ; H1       pickup OK
      AND     M69  ; H2      Pickup  OK
      ANI     M80  ; H1 align completed
      ANI     M81  ; H2 align completed
      ANI     M88  ; H1 load completed
      ANI     M89  ; H2 load completed
      ANI     M91  ; All pick processing
      ANI     M94  ; All Align processing
      ANI     SM400  ; Always ON
      SET     M93  ; Touch   all     Align   Order
594   LD      M103  ; AUTO    RUN
      OR      M150  ; sheet   change  processing
      MPS
      AND     X605  ; Jig detect
      ANI     X600  ; Jig detect
      LDI     X641
      OR      SM400  ; Always ON
      ANB
      SET     Y626  ; CV run control
      MPP
      AND     X600  ; Jig detect
      ANI     M124  ; Touch Lift up
      RST     Y626  ; CV run control
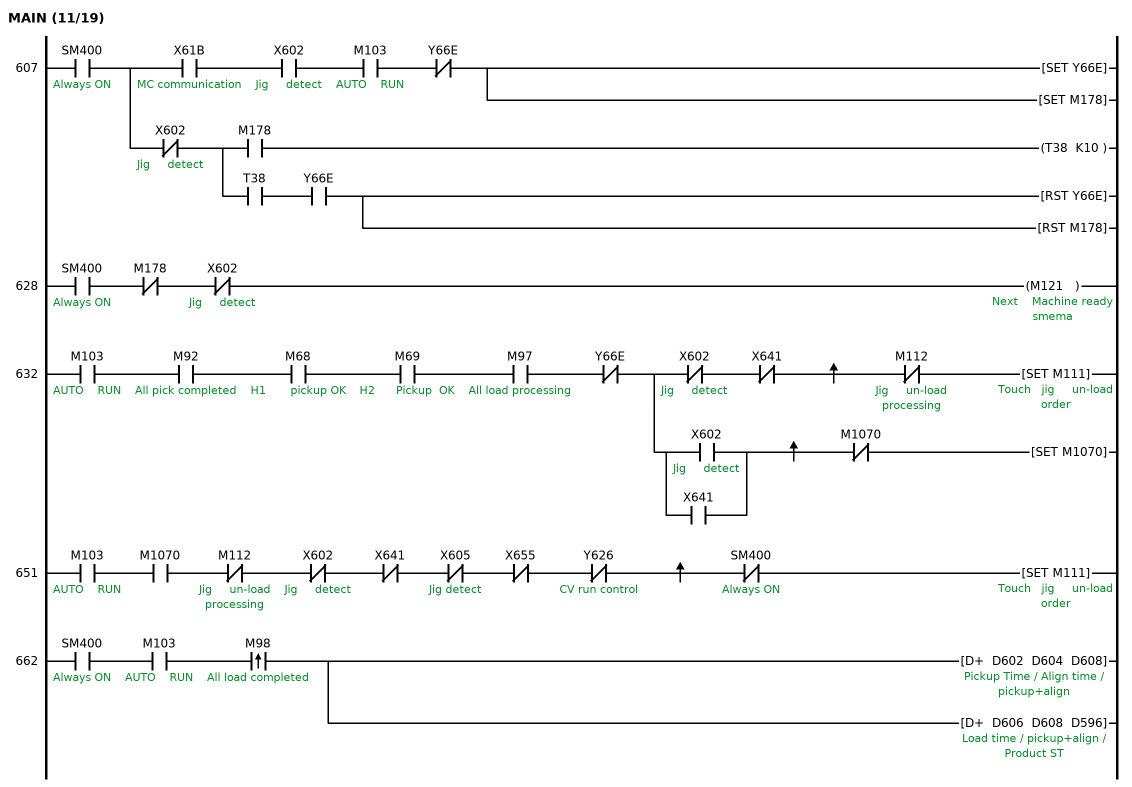
607   LD      SM400  ; Always ON
      MPS
      AND     X61B  ; MC communication
      AND     X602  ; Jig     detect
      AND     M103  ; AUTO    RUN
      ANI     Y66E
      SET     Y66E
      SET     M178
      MPP
      ANI     X602  ; Jig     detect
      MPS
      AND     M178
      OUT     T38 K10
      MPP
      AND     T38
      AND     Y66E
      RST     Y66E
      RST     M178
628   LD      SM400  ; Always ON
      ANI     M178
      ANI     X602  ; Jig     detect
      OUT     M121  ; Next    Machine ready   smema
632   LD      M103  ; AUTO    RUN
      AND     M92  ; All pick completed
      AND     M68  ; H1       pickup OK
      AND     M69  ; H2      Pickup  OK
      AND     M97  ; All load processing
      ANI     Y66E
      MPS
      ANI     X602  ; Jig     detect
      ANI     X641
      MEP
      ANI     M112  ; Jig     un-load processing
      SET     M111  ; Touch   jig     un-load order
      MPP
      LD      X602  ; Jig     detect
      OR      X641
      ANB
      MEP
      ANI     M1070
      SET     M1070
651   LD      M103  ; AUTO    RUN
      AND     M1070
      ANI     M112  ; Jig     un-load processing
      ANI     X602  ; Jig     detect
      ANI     X641
      ANI     X605  ; Jig detect
      ANI     X655
      ANI     Y626  ; CV run control
      MEP
      ANI     SM400  ; Always ON
      SET     M111  ; Touch   jig     un-load order
662   LD      SM400  ; Always ON
      AND     M103  ; AUTO    RUN
      ANDP    M98  ; All load completed
      D+      D602 D604 D608  ; Pickup Time / Align time / pickup+align
      D+      D606 D608 D596  ; Load time / Product ST
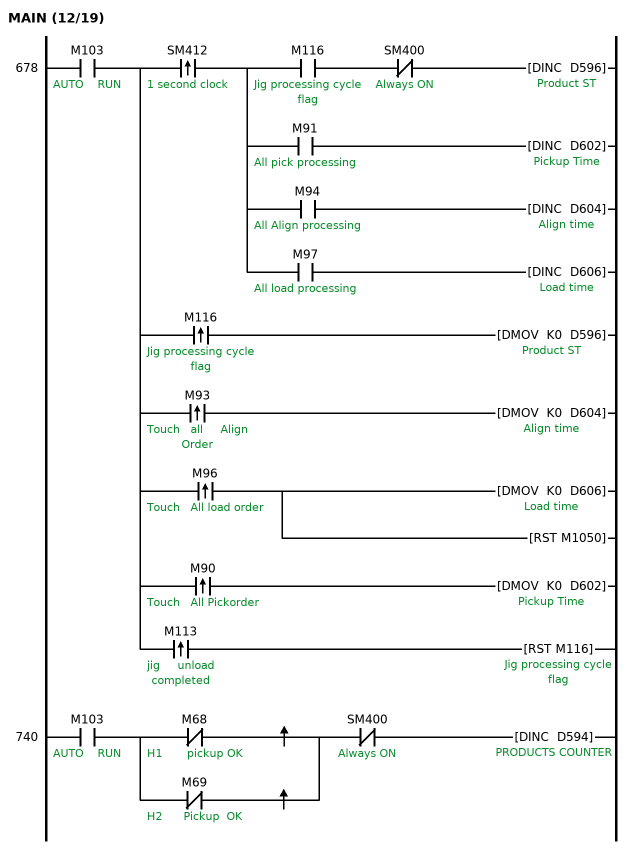
678   LD      M103  ; AUTO    RUN
      MPS
      ANDP    SM412  ; 1 second clock
      MPS
      AND     M116  ; Jig processing cycle flag
      ANI     SM400  ; Always ON
      DINC    D596
      MRD
      AND     M91  ; All pick processing
      DINC    D602
      MRD
      AND     M94  ; All Align processing
      DINC    D604
      MPP
      AND     M97  ; All load processing
      DINC    D606
      MRD
      ANDP    M116  ; Jig processing cycle flag
      DMOV    K0 D596
      MRD
      ANDP    M93  ; Touch   all     Align   Order
      DMOV    K0 D604
      MRD
      ANDP    M96  ; Touch   All load order
      DMOV    K0 D606
      RST     M1050
      MRD
      ANDP    M90  ; Touch   All Pickorder
      DMOV    K0 D602
      MPP
      ANDP    M113  ; jig     unload  completed
      RST     M116  ; Jig processing cycle flag
740   LD      M103  ; AUTO    RUN
      LDI     M68  ; H1       pickup OK
      MEP
      LDI     M69  ; H2      Pickup  OK
      MEP
      ORB
      ANB
      ANI     SM400  ; Always ON
      DINC    D594
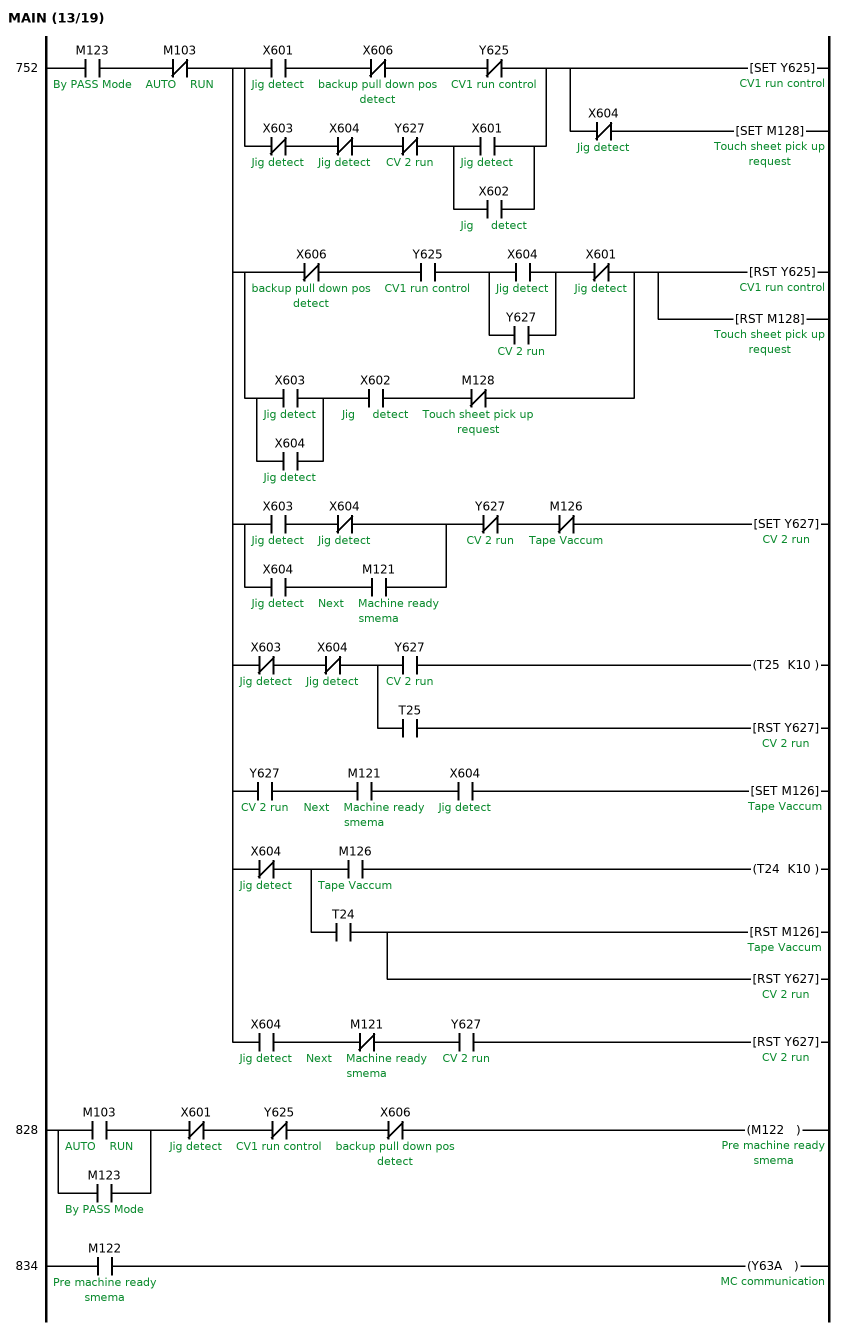
752   LD      M123  ; By PASS Mode
      ANI     M103  ; AUTO    RUN
      MPS
      LD      X601  ; Jig detect
      ANI     X606  ; backup pull down pos detect
      ANI     Y625  ; CV1 run control
      LDI     X603  ; Jig detect
      ANI     X604  ; Jig detect
      ANI     Y627  ; CV 2 run
      LD      X601  ; Jig detect
      OR      X602  ; Jig     detect
      ANB
      ORB
      ANB
      SET     Y625  ; CV1 run control
      ANI     X604  ; Jig detect
      SET     M128  ; Touch sheet pick up request
      MRD
      LDI     X606  ; backup pull down pos detect
      AND     Y625  ; CV1 run control
      LD      X604  ; Jig detect
      OR      Y627  ; CV 2 run
      ANB
      ANI     X601  ; Jig detect
      LD      X603  ; Jig detect
      OR      X604  ; Jig detect
      AND     X602  ; Jig     detect
      ANI     M128  ; Touch sheet pick up request
      ORB
      ANB
      RST     Y625  ; CV1 run control
      RST     M128  ; Touch sheet pick up request
      MRD
      LD      X603  ; Jig detect
      ANI     X604  ; Jig detect
      LD      X604  ; Jig detect
      AND     M121  ; Next    Machine ready   smema
      ORB
      ANB
      ANI     Y627  ; CV 2 run
      ANI     M126  ; Tape Vaccum
      SET     Y627  ; CV 2 run
      MRD
      ANI     X603  ; Jig detect
      ANI     X604  ; Jig detect
      MPS
      AND     Y627  ; CV 2 run
      OUT     T25 K10
      MPP
      AND     T25
      RST     Y627  ; CV 2 run
      MRD
      AND     Y627  ; CV 2 run
      AND     M121  ; Next    Machine ready   smema
      AND     X604  ; Jig detect
      SET     M126  ; Tape Vaccum
      MRD
      ANI     X604  ; Jig detect
      MPS
      AND     M126  ; Tape Vaccum
      OUT     T24 K10
      MPP
      AND     T24
      RST     M126  ; Tape Vaccum
      RST     Y627  ; CV 2 run
      MPP
      AND     X604  ; Jig detect
      ANI     M121  ; Next    Machine ready   smema
      AND     Y627  ; CV 2 run
      RST     Y627  ; CV 2 run
828   LD      M103  ; AUTO    RUN
      OR      M123  ; By PASS Mode
      ANI     X601  ; Jig detect
      ANI     Y625  ; CV1 run control
      ANI     X606  ; backup pull down pos detect
      OUT     M122  ; Pre machine ready smema
834   LD      M122  ; Pre machine ready smema
      OUT     Y63A  ; MC communication
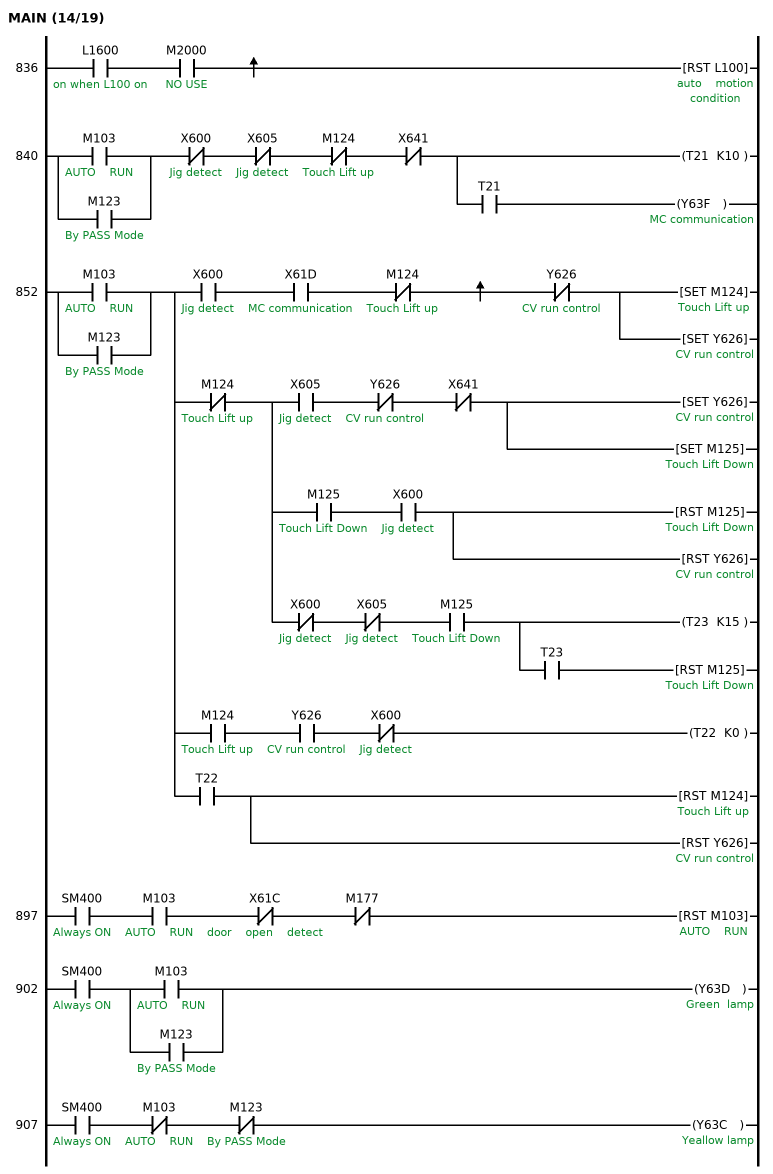
836   LD      L1600  ; on when L100 on
      AND     M2000  ; NO USE
      MEP
      RST     L100  ; auto    motion  condition
840   LD      M103  ; AUTO    RUN
      OR      M123  ; By PASS Mode
      ANI     X600  ; Jig detect
      ANI     X605  ; Jig detect
      ANI     M124  ; Touch Lift up
      ANI     X641
      OUT     T21 K10
      AND     T21
      OUT     Y63F  ; MC communication
852   LD      M103  ; AUTO    RUN
      OR      M123  ; By PASS Mode
      MPS
      AND     X600  ; Jig detect
      AND     X61D  ; MC communication
      ANI     M124  ; Touch Lift up
      MEP
      ANI     Y626  ; CV run control
      SET     M124  ; Touch Lift up
      SET     Y626  ; CV run control
      MRD
      ANI     M124  ; Touch Lift up
      MPS
      AND     X605  ; Jig detect
      ANI     Y626  ; CV run control
      ANI     X641
      SET     Y626  ; CV run control
      SET     M125  ; Touch Lift Down
      MRD
      AND     M125  ; Touch Lift Down
      AND     X600  ; Jig detect
      RST     M125  ; Touch Lift Down
      RST     Y626  ; CV run control
      MPP
      ANI     X600  ; Jig detect
      ANI     X605  ; Jig detect
      AND     M125  ; Touch Lift Down
      OUT     T23 K15
      AND     T23
      RST     M125  ; Touch Lift Down
      MRD
      AND     M124  ; Touch Lift up
      AND     Y626  ; CV run control
      ANI     X600  ; Jig detect
      OUT     T22 K0
      MPP
      AND     T22
      RST     M124  ; Touch Lift up
      RST     Y626  ; CV run control
897   LD      SM400  ; Always ON
      AND     M103  ; AUTO    RUN
      ANI     X61C  ; door    open    detect
      ANI     M177
      RST     M103  ; AUTO    RUN
902   LD      SM400  ; Always ON
      LD      M103  ; AUTO    RUN
      OR      M123  ; By PASS Mode
      ANB
      OUT     Y63D  ; Green  lamp
907   LD      SM400  ; Always ON
      ANI     M103  ; AUTO    RUN
      ANI     M123  ; By PASS Mode
      OUT     Y63C  ; Yeallow lamp
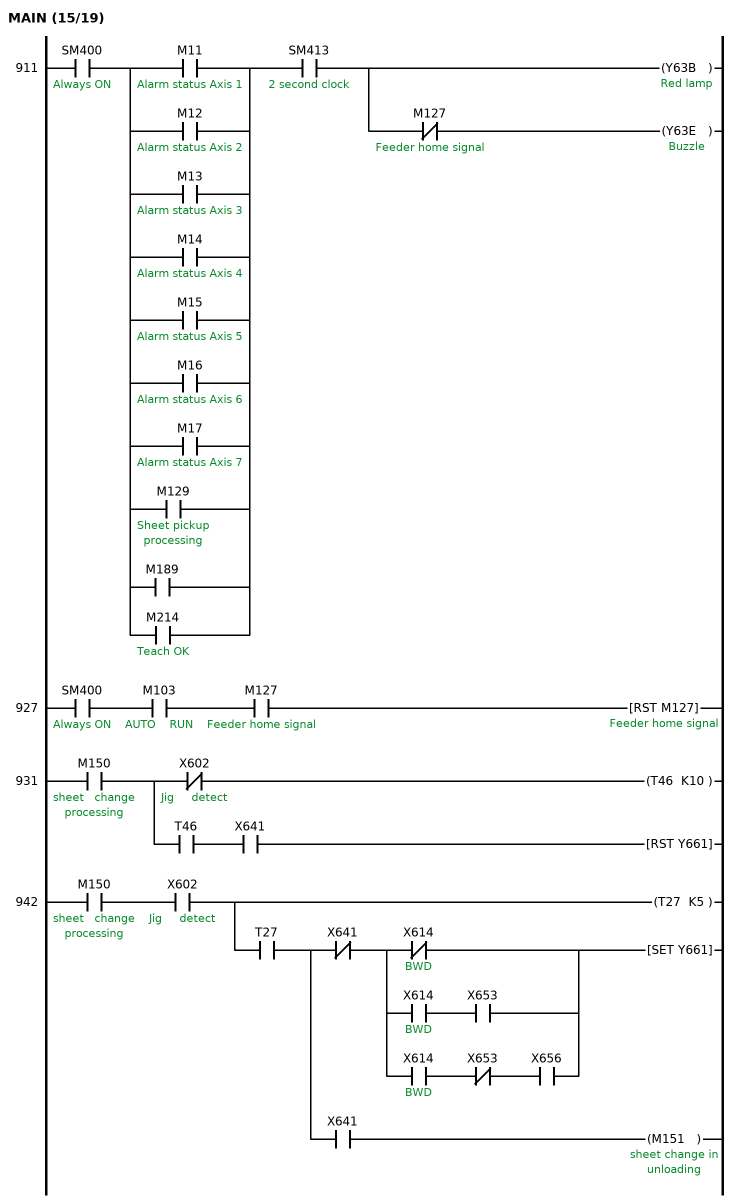
911   LD      SM400  ; Always ON
      LD      M11  ; Alarm status Axis 1
      OR      M12  ; Alarm status Axis 2
      OR      M13  ; Alarm status Axis 3
      OR      M14  ; Alarm status Axis 4
      OR      M15  ; Alarm status Axis 5
      OR      M16  ; Alarm status Axis 6
      OR      M17  ; Alarm status Axis 7
      OR      M129  ; Sheet pickup processing
      OR      M189
      OR      M214  ; Teach OK
      ANB
      AND     SM413  ; 2 second clock
      OUT     Y63B  ; Red lamp
      ANI     M127  ; Feeder home signal
      OUT     Y63E  ; Buzzle
927   LD      SM400  ; Always ON
      AND     M103  ; AUTO    RUN
      AND     M127  ; Feeder home signal
      RST     M127  ; Feeder home signal
931   LD      M150  ; sheet   change  processing
      MPS
      ANI     X602  ; Jig     detect
      OUT     T46 K10
      MPP
      AND     T46
      AND     X641
      RST     Y661
942   LD      M150  ; sheet   change  processing
      AND     X602  ; Jig     detect
      OUT     T27 K5
      AND     T27
      MPS
      ANI     X641
      LDI     X614  ; BWD
      LD      X614  ; BWD
      AND     X653
      ORB
      LD      X614  ; BWD
      ANI     X653
      AND     X656
      ORB
      ANB
      SET     Y661
      MPP
      AND     X641
      OUT     M151  ; sheet change in unloading
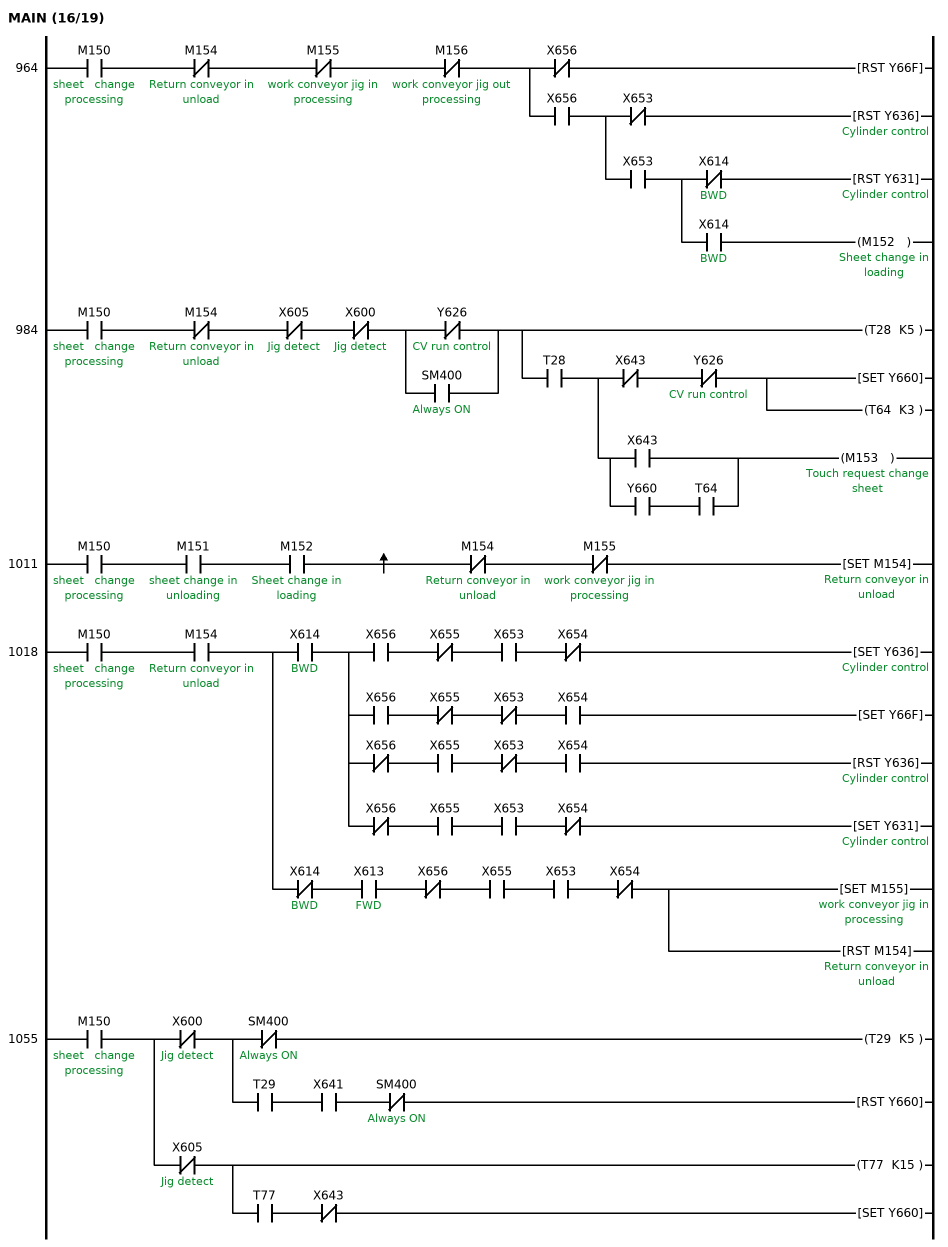
964   LD      M150  ; sheet   change  processing
      ANI     M154  ; Return conveyor in unload
      ANI     M155  ; work conveyor jig in processing
      ANI     M156  ; work conveyor jig out processing
      MPS
      ANI     X656
      RST     Y66F
      MPP
      AND     X656
      MPS
      ANI     X653
      RST     Y636  ; Cylinder control
      MPP
      AND     X653
      MPS
      ANI     X614  ; BWD
      RST     Y631  ; Cylinder control
      MPP
      AND     X614  ; BWD
      OUT     M152  ; Sheet change in loading
984   LD      M150  ; sheet   change  processing
      ANI     M154  ; Return conveyor in unload
      ANI     X605  ; Jig detect
      ANI     X600  ; Jig detect
      LDI     Y626  ; CV run control
      OR      SM400  ; Always ON
      ANB
      OUT     T28 K5
      AND     T28
      MPS
      ANI     X643
      ANI     Y626  ; CV run control
      SET     Y660
      OUT     T64 K3
      MPP
      LD      X643
      LD      Y660
      AND     T64
      ORB
      ANB
      OUT     M153  ; Touch request change sheet
1011  LD      M150  ; sheet   change  processing
      AND     M151  ; sheet change in unloading
      AND     M152  ; Sheet change in loading
      MEP
      ANI     M154  ; Return conveyor in unload
      ANI     M155  ; work conveyor jig in processing
      SET     M154  ; Return conveyor in unload
1018  LD      M150  ; sheet   change  processing
      AND     M154  ; Return conveyor in unload
      MPS
      AND     X614  ; BWD
      MPS
      AND     X656
      ANI     X655
      AND     X653
      ANI     X654
      SET     Y636  ; Cylinder control
      MRD
      AND     X656
      ANI     X655
      ANI     X653
      AND     X654
      SET     Y66F
      MRD
      ANI     X656
      AND     X655
      ANI     X653
      AND     X654
      RST     Y636  ; Cylinder control
      MPP
      ANI     X656
      AND     X655
      AND     X653
      ANI     X654
      SET     Y631  ; Cylinder control
      MPP
      ANI     X614  ; BWD
      AND     X613  ; FWD
      ANI     X656
      AND     X655
      AND     X653
      ANI     X654
      SET     M155  ; work conveyor jig in processing
      RST     M154  ; Return conveyor in unload
1055  LD      M150  ; sheet   change  processing
      MPS
      ANI     X600  ; Jig detect
      MPS
      ANI     SM400  ; Always ON
      OUT     T29 K5
      MPP
      AND     T29
      AND     X641
      ANI     SM400  ; Always ON
      RST     Y660
      MPP
      ANI     X605  ; Jig detect
      OUT     T77 K15
      AND     T77
      ANI     X643
      SET     Y660
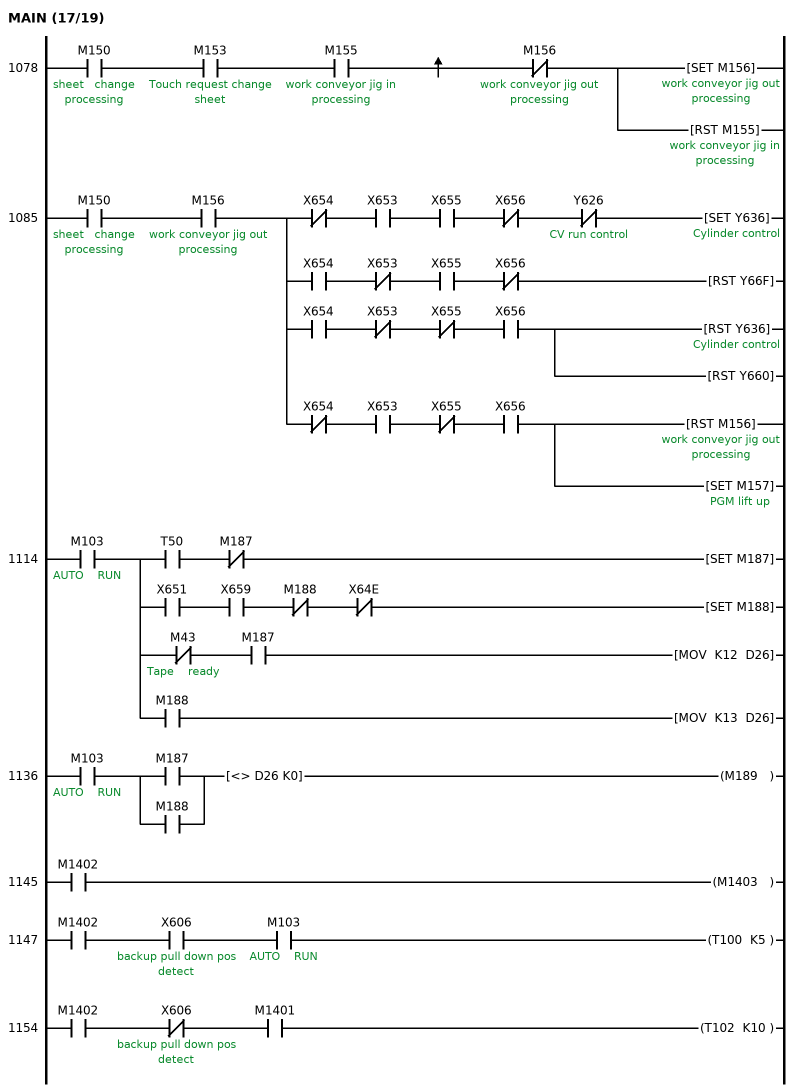
1078  LD      M150  ; sheet   change  processing
      AND     M153  ; Touch request change sheet
      AND     M155  ; work conveyor jig in processing
      MEP
      ANI     M156  ; work conveyor jig out processing
      SET     M156  ; work conveyor jig out processing
      RST     M155  ; work conveyor jig in processing
1085  LD      M150  ; sheet   change  processing
      AND     M156  ; work conveyor jig out processing
      MPS
      ANI     X654
      AND     X653
      AND     X655
      ANI     X656
      ANI     Y626  ; CV run control
      SET     Y636  ; Cylinder control
      MRD
      AND     X654
      ANI     X653
      AND     X655
      ANI     X656
      RST     Y66F
      MRD
      AND     X654
      ANI     X653
      ANI     X655
      AND     X656
      RST     Y636  ; Cylinder control
      RST     Y660
      MPP
      ANI     X654
      AND     X653
      ANI     X655
      AND     X656
      RST     M156  ; work conveyor jig out processing
      SET     M157  ; PGM lift up
1114  LD      M103  ; AUTO    RUN
      MPS
      AND     T50
      ANI     M187
      SET     M187
      MRD
      AND     X651
      AND     X659
      ANI     M188
      ANI     X64E
      SET     M188
      MRD
      ANI     M43  ; Tape    ready
      AND     M187
      MOV     K12 D26
      MPP
      AND     M188
      MOV     K13 D26
1136  LD      M103  ; AUTO    RUN
      LD      M187
      OR      M188
      ANB
      AND<>   D26 K0
      OUT     M189
1145  LD      M1402
      OUT     M1403
1147  LD      M1402
      AND     X606  ; backup pull down pos detect
      AND     M103  ; AUTO    RUN
      OUT     T100 K5
1154  LD      M1402
      ANI     X606  ; backup pull down pos detect
      AND     M1401
      OUT     T102 K10
